LIN {X 0,Y 348.002,Z 736.138,A -85,B 0,C 180,E1 -13689.297,E2 -13689.297} C_VEL
LIN {X 0,Y 349.039,Z 729.917,A -85,B 0,C 180,E1 -13691.322,E2 -13691.322} C_VEL
LIN {X 0,Y 350.021,Z 723.137,A -85,B 0,C 180,E1 -13693.055,E2 -13693.055} C_VEL
LIN {X 0,Y 351.346,Z 714.648,A -85,B 0,C 180,E1 -13694.776,E2 -13694.776} C_VEL
LIN {X 0,Y 352.644,Z 705.984,A -85,B 0,C 180,E1 -13696.201,E2 -13696.201} C_VEL
LIN {X 0,Y 354,Z 696.385,A -85,B 0,C 180,E1 -13697.489,E2 -13697.489} C_VEL
LIN {X 0,Y 355.527,Z 683.397,A -85,B 0,C 180,E1 -13698.887,E2 -13698.887} C_VEL
LIN {X 0,Y 356.754,Z 671.65,A -85,B 0,C 180,E1 -13699.866,E2 -13699.866} C_VEL
LIN {X 0,Y 357.956,Z 658.586,A -85,B 0,C 180,E1 -13700.696,E2 -13700.696} C_VEL
LIN {X 0,Y 358.841,Z 645.608,A -85,B 0,C 180,E1 -13701.281,E2 -13701.281} C_VEL
LIN {X 0,Y 363.919,Z 560.799,A -85,B 0,C 180,E1 -13703.957,E2 -13703.957} C_VEL
LIN {X 0,Y 363.845,Z 556.971,A -85,B 0,C 180,E1 -13704.121,E2 -13704.121} C_VEL
LIN {X 0,Y 360.997,Z 542.499,A -85,B 0,C 180,E1 -13705.115,E2 -13705.115} C_VEL
LIN {X 0,Y 359.502,Z 536.273,A -85,B 0,C 180,E1 -13705.621,E2 -13705.621} C_VEL
LIN {X 0,Y 361.494,Z 519.718,A -85,B 0,C 180,E1 -13708.755,E2 -13708.755} C_VEL
LIN {X 0,Y 360.696,Z 513.547,A -85,B 0,C 180,E1 -13710.252,E2 -13710.252} C_VEL
LIN {X 0,Y 358.682,Z 505.189,A -85,B 0,C 180,E1 -13712.589,E2 -13712.589} C_VEL
LIN {X 0,Y 356.57,Z 498.193,A -85,B 0,C 180,E1 -13714.861,E2 -13714.861} C_VEL
LIN {X 0,Y 353.95,Z 491.68,A -85,B 0,C 180,E1 -13717.415,E2 -13717.415} C_VEL
LIN {X 0,Y 351.895,Z 487.111,A -85,B 0,C 180,E1 -13719.725,E2 -13719.725} C_VEL
LIN {X 0,Y 350.344,Z 483.44,A -85,B 0,C 180,E1 -13722.077,E2 -13722.077} C_VEL
LIN {X 0,Y 348.527,Z 481.325,A -85,B 0,C 180,E1 -13725.107,E2 -13725.107} C_VEL
LIN {X 0,Y 348.251,Z 480.7,A -85,B 0,C 180,E1 -13726.673,E2 -13726.673} C_VEL
LIN {X 0,Y 348.29,Z 480.742,A -85,B 0,C 180,E1 -13728.297,E2 -13728.297} C_VEL
LIN {X 0,Y 348.675,Z 481.499,A -85,B 0,C 180,E1 -13729.991,E2 -13729.991} C_VEL
LIN {X 0,Y 349.596,Z 482.735,A -85,B 0,C 180,E1 -13731.631,E2 -13731.631} C_VEL
LIN {X 0,Y 351.074,Z 484.356,A -85,B 0,C 180,E1 -13733.201,E2 -13733.201} C_VEL
LIN {X 0,Y 352.123,Z 487.497,A -85,B 0,C 180,E1 -13734.632,E2 -13734.632} C_VEL
LIN {X 0,Y 352.81,Z 490.868,A -85,B 0,C 180,E1 -13735.683,E2 -13735.683} C_VEL
LIN {X 0,Y 355.082,Z 501.742,A -85,B 0,C 180,E1 -13738.329,E2 -13738.329} C_VEL
LIN {X 0,Y 357.463,Z 510.29,A -85,B 0,C 180,E1 -13740.056,E2 -13740.056} C_VEL
LIN {X 0,Y 358.938,Z 516.196,A -85,B 0,C 180,E1 -13741.042,E2 -13741.042} C_VEL
LIN {X 0,Y 359.355,Z 523.121,A -85,B 0,C 180,E1 -13741.84,E2 -13741.84} C_VEL
LIN {X 0,Y 359.68,Z 533.701,A -85,B 0,C 180,E1 -13742.9,E2 -13742.9} C_VEL
LIN {X 0,Y 359.381,Z 549.497,A -85,B 0,C 180,E1 -13744.142,E2 -13744.142} C_VEL
LIN {X 0,Y 360.003,Z 556.284,A -85,B 0,C 180,E1 -13744.341,E2 -13744.341} C_VEL
LIN {X 0,Y 357.565,Z 655.14,A -85,B 0,C 180,E1 -13746.468,E2 -13746.468} C_VEL
LIN {X 0,Y 356.73,Z 669.286,A -85,B 0,C 180,E1 -13746.985,E2 -13746.985} C_VEL
LIN {X 0,Y 355.576,Z 683.012,A -85,B 0,C 180,E1 -13747.712,E2 -13747.712} C_VEL
LIN {X 0,Y 354.434,Z 695.886,A -85,B 0,C 180,E1 -13748.631,E2 -13748.631} C_VEL
LIN {X 0,Y 353.249,Z 707.122,A -85,B 0,C 180,E1 -13749.64,E2 -13749.64} C_VEL
LIN {X 0,Y 351.889,Z 718.658,A -85,B 0,C 180,E1 -13750.909,E2 -13750.909} C_VEL
LIN {X 0,Y 350.595,Z 728.367,A -85,B 0,C 180,E1 -13752.198,E2 -13752.198} C_VEL
LIN {X 0,Y 349.238,Z 739.157,A -85,B 0,C 180,E1 -13753.935,E2 -13753.935} C_VEL
LIN {X 0,Y 348.218,Z 747.853,A -85,B 0,C 180,E1 -13755.644,E2 -13755.644} C_VEL
LIN {X 0,Y 347.489,Z 755.405,A -85,B 0,C 180,E1 -13757.441,E2 -13757.441} C_VEL
LIN {X 0,Y 346.772,Z 762.421,A -85,B 0,C 180,E1 -13759.489,E2 -13759.489} C_VEL
LIN {X 0,Y 346.391,Z 768.747,A -85,B 0,C 180,E1 -13761.834,E2 -13761.834} C_VEL
LIN {X 0,Y 346.287,Z 773.108,A -85,B 0,C 180,E1 -13763.971,E2 -13763.971} C_VEL
LIN {X 0,Y 346.266,Z 775.106,A -85,B 0,C 180,E1 -13765.342,E2 -13765.342} C_VEL
LIN {X 0,Y 346.234,Z 776.287,A -85,B 0,C 180,E1 -13766.507,E2 -13766.507} C_VEL
LIN {X 0,Y 346.383,Z 777.549,A -85,B 0,C 180,E1 -13768.836,E2 -13768.836} C_VEL
LIN {X 0,Y 346.383,Z 777.546,A -85,B 0,C 180,E1 -13771.161,E2 -13771.161} C_VEL
LIN {X 0,Y 346.234,Z 776.058,A -85,B 0,C 180,E1 -13773.49,E2 -13773.49} C_VEL
LIN {X 0,Y 346.268,Z 774.768,A -85,B 0,C 180,E1 -13774.655,E2 -13774.655} C_VEL
LIN {X 0,Y 346.323,Z 772.679,A -85,B 0,C 180,E1 -13776.085,E2 -13776.085} C_VEL
LIN {X 0,Y 346.388,Z 768.585,A -85,B 0,C 180,E1 -13778.163,E2 -13778.163} C_VEL
LIN {X 0,Y 346.647,Z 764.085,A -85,B 0,C 180,E1 -13779.922,E2 -13779.922} C_VEL
LIN {X 0,Y 347.28,Z 757.517,A -85,B 0,C 180,E1 -13781.97,E2 -13781.97} C_VEL
LIN {X 0,Y 347.93,Z 750.584,A -85,B 0,C 180,E1 -13783.728,E2 -13783.728} C_VEL
LIN {X 0,Y 348.883,Z 742.235,A -85,B 0,C 180,E1 -13785.479,E2 -13785.479} C_VEL
LIN {X 0,Y 350.113,Z 732.148,A -85,B 0,C 180,E1 -13787.221,E2 -13787.221} C_VEL
LIN {X 0,Y 351.394,Z 722.009,A -85,B 0,C 180,E1 -13788.661,E2 -13788.661} C_VEL
LIN {X 0,Y 352.753,Z 711.083,A -85,B 0,C 180,E1 -13789.944,E2 -13789.944} C_VEL
LIN {X 0,Y 353.991,Z 699.35,A -85,B 0,C 180,E1 -13791.073,E2 -13791.073} C_VEL
LIN {X 0,Y 355.335,Z 686.208,A -85,B 0,C 180,E1 -13792.071,E2 -13792.071} C_VEL
LIN {X 0,Y 356.479,Z 672.058,A -85,B 0,C 180,E1 -13792.875,E2 -13792.875} C_VEL
LIN {X 0,Y 357.403,Z 658.122,A -85,B 0,C 180,E1 -13793.425,E2 -13793.425} C_VEL
LIN {X 0,Y 358.032,Z 637.673,A -85,B 0,C 180,E1 -13793.919,E2 -13793.919} C_VEL
LIN {X 0,Y 359.927,Z 554.026,A -85,B 0,C 180,E1 -13795.701,E2 -13795.701} C_VEL
LIN {X 0,Y 355.225,Z 521.927,A -85,B 0,C 180,E1 -13796.777,E2 -13796.777} C_VEL
LIN {X 0,Y 356.403,Z 514.04,A -85,B 0,C 180,E1 -13798.244,E2 -13798.244} C_VEL
LIN {X 0,Y 355.634,Z 509.249,A -85,B 0,C 180,E1 -13799.261,E2 -13799.261} C_VEL
LIN {X 0,Y 352.934,Z 497.682,A -85,B 0,C 180,E1 -13801.847,E2 -13801.847} C_VEL
LIN {X 0,Y 349.447,Z 484.664,A -85,B 0,C 180,E1 -13804.936,E2 -13804.936} C_VEL
LIN {X 0,Y 347.764,Z 478.78,A -85,B 0,C 180,E1 -13806.471,E2 -13806.471} C_VEL
LIN {X 0,Y 347.786,Z 478.79,A -85,B 0,C 180,E1 -13810.287,E2 -13810.287} C_VEL
LIN {X 0,Y 347.811,Z 478.784,A -85,B 0,C 180,E1 -13813.392,E2 -13813.392} C_VEL
LIN {X 0,Y 347.81,Z 478.786,A -85,B 0,C 180,E1 -13816.669,E2 -13816.669} C_VEL
LIN {X 0,Y 347.777,Z 478.783,A -85,B 0,C 180,E1 -13820.164,E2 -13820.164} C_VEL
LIN {X 0,Y 347.78,Z 478.764,A -85,B 0,C 180,E1 -13824.124,E2 -13824.124} C_VEL
LIN {X 0,Y 347.754,Z 478.787,A -85,B 0,C 180,E1 -13828.301,E2 -13828.301} C_VEL
LIN {X 0,Y 347.796,Z 478.785,A -85,B 0,C 180,E1 -13830.989,E2 -13830.989} C_VEL
LIN {X 0,Y 347.821,Z 478.782,A -85,B 0,C 180,E1 -13833.607,E2 -13833.607} C_VEL
LIN {X 0,Y 347.777,Z 478.774,A -85,B 0,C 180,E1 -13836.161,E2 -13836.161} C_VEL
LIN {X 0,Y 347.796,Z 478.774,A -85,B 0,C 180,E1 -13839.908,E2 -13839.908} C_VEL
LIN {X 0,Y 347.855,Z 478.781,A -85,B 0,C 180,E1 -13842.359,E2 -13842.359} C_VEL
LIN {X 0,Y 347.886,Z 478.773,A -85,B 0,C 180,E1 -13845.97,E2 -13845.97} C_VEL
LIN {X 0,Y 347.922,Z 478.765,A -85,B 0,C 180,E1 -13849.526,E2 -13849.526} C_VEL
LIN {X 0,Y 348.063,Z 478.752,A -85,B 0,C 180,E1 -13851.875,E2 -13851.875} C_VEL
LIN {X 0,Y 348.058,Z 478.744,A -85,B 0,C 180,E1 -13854.206,E2 -13854.206} C_VEL
LIN {X 0,Y 348.198,Z 478.731,A -85,B 0,C 180,E1 -13857.687,E2 -13857.687} C_VEL
LIN {X 0,Y 348.358,Z 478.713,A -85,B 0,C 180,E1 -13860,E2 -13860} C_VEL
LIN {X 0,Y 348.198,Z 478.734,A -85,B 0,C 180,E1 -13862.314,E2 -13862.314} C_VEL
LIN {X 0,Y 348.095,Z 478.746,A -85,B 0,C 180,E1 -13866.958,E2 -13866.958} C_VEL
LIN {X 0,Y 347.958,Z 478.762,A -85,B 0,C 180,E1 -13869.299,E2 -13869.299} C_VEL
LIN {X 0,Y 347.883,Z 478.767,A -85,B 0,C 180,E1 -13872.84,E2 -13872.84} C_VEL
LIN {X 0,Y 347.831,Z 478.782,A -85,B 0,C 180,E1 -13876.432,E2 -13876.432} C_VEL
LIN {X 0,Y 347.846,Z 478.778,A -85,B 0,C 180,E1 -13878.861,E2 -13878.861} C_VEL
LIN {X 0,Y 347.764,Z 478.785,A -85,B 0,C 180,E1 -13882.58,E2 -13882.58} C_VEL
LIN {X 0,Y 347.802,Z 478.783,A -85,B 0,C 180,E1 -13885.109,E2 -13885.109} C_VEL
LIN {X 0,Y 347.803,Z 478.783,A -85,B 0,C 180,E1 -13887.695,E2 -13887.695} C_VEL
LIN {X 0,Y 347.762,Z 478.785,A -85,B 0,C 180,E1 -13890.347,E2 -13890.347} C_VEL
LIN {X 0,Y 347.754,Z 478.786,A -85,B 0,C 180,E1 -13894.049,E2 -13894.049} C_VEL
LIN {X 0,Y 347.756,Z 478.787,A -85,B 0,C 180,E1 -13897.322,E2 -13897.322} C_VEL
LIN {X 0,Y 347.748,Z 478.791,A -85,B 0,C 180,E1 -13900.295,E2 -13900.295} C_VEL
LIN {X 0,Y 347.762,Z 478.789,A -85,B 0,C 180,E1 -13903.402,E2 -13903.402} C_VEL
LIN {X 0,Y 347.779,Z 478.792,A -85,B 0,C 180,E1 -13906.677,E2 -13906.677} C_VEL
LIN {X 0,Y 347.78,Z 478.788,A -85,B 0,C 180,E1 -13910.167,E2 -13910.167} C_VEL
LIN {X 0,Y 347.785,Z 478.785,A -85,B 0,C 180,E1 -13914.127,E2 -13914.127} C_VEL
LIN {X 0,Y 347.774,Z 478.899,A -85,B 0,C 180,E1 -13916.323,E2 -13916.323} C_VEL
LIN {X 0,Y 350.302,Z 488.761,A -85,B 0,C 180,E1 -13919.151,E2 -13919.151} C_VEL
LIN {X 0,Y 352.862,Z 499.54,A -85,B 0,C 180,E1 -13922.094,E2 -13922.094} C_VEL
LIN {X 0,Y 354.273,Z 507.484,A -85,B 0,C 180,E1 -13924.126,E2 -13924.126} C_VEL
LIN {X 0,Y 353.241,Z 516.92,A -85,B 0,C 180,E1 -13926.236,E2 -13926.236} C_VEL
LIN {X 0,Y 358.606,Z 543.403,A -85,B 0,C 180,E1 -13927.182,E2 -13927.182} C_VEL
LIN {X 0,Y 359.417,Z 548.206,A -85,B 0,C 180,E1 -13927.337,E2 -13927.337} C_VEL
LIN {X 0,Y 358.007,Z 631.224,A -85,B 0,C 180,E1 -13928.895,E2 -13928.895} C_VEL
LIN {X 0,Y 357.474,Z 644.098,A -85,B 0,C 180,E1 -13929.352,E2 -13929.352} C_VEL
LIN {X 0,Y 356.593,Z 657.19,A -85,B 0,C 180,E1 -13930.051,E2 -13930.051} C_VEL
LIN {X 0,Y 355.469,Z 669.587,A -85,B 0,C 180,E1 -13930.962,E2 -13930.962} C_VEL
LIN {X 0,Y 354.252,Z 681.206,A -85,B 0,C 180,E1 -13932.093,E2 -13932.093} C_VEL
LIN {X 0,Y 353.116,Z 690.811,A -85,B 0,C 180,E1 -13933.261,E2 -13933.261} C_VEL
LIN {X 0,Y 351.728,Z 700.18,A -85,B 0,C 180,E1 -13934.649,E2 -13934.649} C_VEL
LIN {X 0,Y 350.417,Z 709.509,A -85,B 0,C 180,E1 -13936.371,E2 -13936.371} C_VEL
LIN {X 0,Y 349.322,Z 716.98,A -85,B 0,C 180,E1 -13938.101,E2 -13938.101} C_VEL
LIN {X 0,Y 348.184,Z 723.886,A -85,B 0,C 180,E1 -13940.122,E2 -13940.122} C_VEL
LIN {X 0,Y 347.475,Z 728.531,A -85,B 0,C 180,E1 -13941.862,E2 -13941.862} C_VEL
LIN {X 0,Y 347.067,Z 732.133,A -85,B 0,C 180,E1 -13943.607,E2 -13943.607} C_VEL
LIN {X 0,Y 346.68,Z 734.808,A -85,B 0,C 180,E1 -13945.35,E2 -13945.35} C_VEL
LIN {X 0,Y 346.546,Z 736.986,A -85,B 0,C 180,E1 -13947.677,E2 -13947.677} C_VEL
LIN {X 0,Y 346.395,Z 737.758,A -85,B 0,C 180,E1 -13950.002,E2 -13950.002} C_VEL
LIN {X 0,Y 346.545,Z 737.05,A -85,B 0,C 180,E1 -13952.326,E2 -13952.326} C_VEL
LIN {X 0,Y 346.653,Z 734.923,A -85,B 0,C 180,E1 -13954.653,E2 -13954.653} C_VEL
LIN {X 0,Y 347.06,Z 732.305,A -85,B 0,C 180,E1 -13956.396,E2 -13956.396} C_VEL
LIN {X 0,Y 347.477,Z 728.765,A -85,B 0,C 180,E1 -13958.141,E2 -13958.141} C_VEL
LIN {X 0,Y 348.138,Z 724.186,A -85,B 0,C 180,E1 -13959.882,E2 -13959.882} C_VEL
LIN {X 0,Y 349.206,Z 717.352,A -85,B 0,C 180,E1 -13961.906,E2 -13961.906} C_VEL
LIN {X 0,Y 350.404,Z 709.975,A -85,B 0,C 180,E1 -13963.632,E2 -13963.632} C_VEL
LIN {X 0,Y 351.457,Z 702.468,A -85,B 0,C 180,E1 -13965.069,E2 -13965.069} C_VEL
LIN {X 0,Y 352.73,Z 693.648,A -85,B 0,C 180,E1 -13966.457,E2 -13966.457} C_VEL
LIN {X 0,Y 353.963,Z 683.345,A -85,B 0,C 180,E1 -13967.775,E2 -13967.775} C_VEL
LIN {X 0,Y 355.25,Z 672.22,A -85,B 0,C 180,E1 -13968.903,E2 -13968.903} C_VEL
LIN {X 0,Y 356.257,Z 661.72,A -85,B 0,C 180,E1 -13969.746,E2 -13969.746} C_VEL
LIN {X 0,Y 357.22,Z 649.066,A -85,B 0,C 180,E1 -13970.516,E2 -13970.516} C_VEL
LIN {X 0,Y 357.878,Z 636.708,A -85,B 0,C 180,E1 -13971.041,E2 -13971.041} C_VEL
LIN {X 0,Y 358.257,Z 622.461,A -85,B 0,C 180,E1 -13971.394,E2 -13971.394} C_VEL
LIN {X 0,Y 358.873,Z 586.038,A -85,B 0,C 180,E1 -13972.062,E2 -13972.062} C_VEL
LIN {X 0,Y 358.321,Z 580.227,A -85,B 0,C 180,E1 -13972.214,E2 -13972.214} C_VEL
LIN {X 0,Y 353.289,Z 561.575,A -85,B 0,C 180,E1 -13972.947,E2 -13972.947} C_VEL
LIN {X 0,Y 352.843,Z 555.764,A -85,B 0,C 180,E1 -13973.098,E2 -13973.098} C_VEL
LIN {X 0,Y 352.748,Z 547.495,A -85,B 0,C 180,E1 -13973.274,E2 -13973.274} C_VEL
LIN {X 0,Y 347.839,Z 522.801,A -85,B 0,C 180,E1 -13974.169,E2 -13974.169} C_VEL
LIN {X 0,Y 346.602,Z 516.839,A -85,B 0,C 180,E1 -13974.4,E2 -13974.4} C_VEL
LIN {X 0,Y 347.445,Z 509.457,A -85,B 0,C 180,E1 -13976.102,E2 -13976.102} C_VEL
LIN {X 0,Y 345.815,Z 500.603,A -85,B 0,C 180,E1 -13978.42,E2 -13978.42} C_VEL
LIN {X 0,Y 343.291,Z 489.688,A -85,B 0,C 180,E1 -13981.47,E2 -13981.47} C_VEL
LIN {X 0,Y 340.716,Z 479.667,A -85,B 0,C 180,E1 -13984.476,E2 -13984.476} C_VEL
LIN {X 0,Y 340.718,Z 479.665,A -85,B 0,C 180,E1 -13988.387,E2 -13988.387} C_VEL
LIN {X 0,Y 340.706,Z 479.67,A -85,B 0,C 180,E1 -13992.046,E2 -13992.046} C_VEL
LIN {X 0,Y 340.659,Z 479.676,A -85,B 0,C 180,E1 -13996.227,E2 -13996.227} C_VEL
LIN {X 0,Y 340.695,Z 479.674,A -85,B 0,C 180,E1 -13999.753,E2 -13999.753} C_VEL
LIN {X 0,Y 340.712,Z 479.663,A -85,B 0,C 180,E1 -14003.259,E2 -14003.259} C_VEL
LIN {X 0,Y 340.701,Z 479.672,A -85,B 0,C 180,E1 -14006.154,E2 -14006.154} C_VEL
LIN {X 0,Y 340.717,Z 479.682,A -85,B 0,C 180,E1 -14008.352,E2 -14008.352} C_VEL
LIN {X 0,Y 344.486,Z 495.918,A -85,B 0,C 180,E1 -14011.629,E2 -14011.629} C_VEL
LIN {X 0,Y 346.265,Z 505.327,A -85,B 0,C 180,E1 -14013.479,E2 -14013.479} C_VEL
LIN {X 0,Y 345.11,Z 524.906,A -85,B 0,C 180,E1 -14017.003,E2 -14017.003} C_VEL
LIN {X 0,Y 344.655,Z 531.676,A -85,B 0,C 180,E1 -14018.211,E2 -14018.211} C_VEL
LIN {X 0,Y 347.781,Z 555.235,A -85,B 0,C 180,E1 -14019.034,E2 -14019.034} C_VEL
LIN {X 0,Y 345.289,Z 643.42,A -85,B 0,C 180,E1 -14021.494,E2 -14021.494} C_VEL
LIN {X 0,Y 344.768,Z 655.803,A -85,B 0,C 180,E1 -14022.042,E2 -14022.042} C_VEL
LIN {X 0,Y 344.12,Z 669.789,A -85,B 0,C 180,E1 -14022.927,E2 -14022.927} C_VEL
LIN {X 0,Y 343.327,Z 682.066,A -85,B 0,C 180,E1 -14023.958,E2 -14023.958} C_VEL
LIN {X 0,Y 342.562,Z 694.465,A -85,B 0,C 180,E1 -14025.292,E2 -14025.292} C_VEL
LIN {X 0,Y 341.764,Z 704.362,A -85,B 0,C 180,E1 -14026.624,E2 -14026.624} C_VEL
LIN {X 0,Y 341,Z 713.429,A -85,B 0,C 180,E1 -14028.106,E2 -14028.106} C_VEL
LIN {X 0,Y 340.474,Z 720.954,A -85,B 0,C 180,E1 -14029.594,E2 -14029.594} C_VEL
LIN {X 0,Y 339.947,Z 728.322,A -85,B 0,C 180,E1 -14031.38,E2 -14031.38} C_VEL
LIN {X 0,Y 339.566,Z 734.985,A -85,B 0,C 180,E1 -14033.45,E2 -14033.45} C_VEL
LIN {X 0,Y 339.373,Z 739.411,A -85,B 0,C 180,E1 -14035.248,E2 -14035.248} C_VEL
LIN {X 0,Y 339.25,Z 741.676,A -85,B 0,C 180,E1 -14036.437,E2 -14036.437} C_VEL
LIN {X 0,Y 339.179,Z 743.473,A -85,B 0,C 180,E1 -14037.625,E2 -14037.625} C_VEL
LIN {X 0,Y 339.182,Z 744.84,A -85,B 0,C 180,E1 -14038.813,E2 -14038.813} C_VEL
LIN {X 0,Y 339.194,Z 745.719,A -85,B 0,C 180,E1 -14040,E2 -14040} C_VEL
LIN {X 0,Y 339.298,Z 746.17,A -85,B 0,C 180,E1 -14041.187,E2 -14041.187} C_VEL
LIN {X 0,Y 339.445,Z 746.207,A -85,B 0,C 180,E1 -14042.373,E2 -14042.373} C_VEL
LIN {X 0,Y 339.551,Z 745.781,A -85,B 0,C 180,E1 -14043.56,E2 -14043.56} C_VEL
LIN {X 0,Y 339.598,Z 744.931,A -85,B 0,C 180,E1 -14044.748,E2 -14044.748} C_VEL
LIN {X 0,Y 339.805,Z 743.66,A -85,B 0,C 180,E1 -14045.936,E2 -14045.936} C_VEL
LIN {X 0,Y 340.457,Z 740.793,A -85,B 0,C 180,E1 -14047.747,E2 -14047.747} C_VEL
LIN {X 0,Y 341.06,Z 736.982,A -85,B 0,C 180,E1 -14049.488,E2 -14049.488} C_VEL
LIN {X 0,Y 342,Z 731.922,A -85,B 0,C 180,E1 -14051.258,E2 -14051.258} C_VEL
LIN {X 0,Y 343.04,Z 725.521,A -85,B 0,C 180,E1 -14053.024,E2 -14053.024} C_VEL
LIN {X 0,Y 344.404,Z 717.548,A -85,B 0,C 180,E1 -14054.778,E2 -14054.778} C_VEL
LIN {X 0,Y 345.72,Z 709.388,A -85,B 0,C 180,E1 -14056.231,E2 -14056.231} C_VEL
LIN {X 0,Y 347.283,Z 699.489,A -85,B 0,C 180,E1 -14057.671,E2 -14057.671} C_VEL
LIN {X 0,Y 348.747,Z 688.6,A -85,B 0,C 180,E1 -14058.963,E2 -14058.963} C_VEL
LIN {X 0,Y 349.989,Z 678.066,A -85,B 0,C 180,E1 -14059.96,E2 -14059.96} C_VEL
LIN {X 0,Y 351.248,Z 665.724,A -85,B 0,C 180,E1 -14060.879,E2 -14060.879} C_VEL
LIN {X 0,Y 352.423,Z 651.807,A -85,B 0,C 180,E1 -14061.649,E2 -14061.649} C_VEL
LIN {X 0,Y 353.379,Z 636.861,A -85,B 0,C 180,E1 -14062.202,E2 -14062.202} C_VEL
LIN {X 0,Y 357.783,Z 569.211,A -85,B 0,C 180,E1 -14064.401,E2 -14064.401} C_VEL
LIN {X 0,Y 358.449,Z 559.585,A -85,B 0,C 180,E1 -14064.725,E2 -14064.725} C_VEL
LIN {X 0,Y 355.835,Z 545.585,A -85,B 0,C 180,E1 -14065.719,E2 -14065.719} C_VEL
LIN {X 0,Y 353.816,Z 536.839,A -85,B 0,C 180,E1 -14066.461,E2 -14066.461} C_VEL
LIN {X 0,Y 355.596,Z 523.958,A -85,B 0,C 180,E1 -14068.946,E2 -14068.946} C_VEL
LIN {X 0,Y 355.39,Z 519.767,A -85,B 0,C 180,E1 -14069.909,E2 -14069.909} C_VEL
LIN {X 0,Y 353.845,Z 511.889,A -85,B 0,C 180,E1 -14072.093,E2 -14072.093} C_VEL
LIN {X 0,Y 351.449,Z 503.214,A -85,B 0,C 180,E1 -14074.925,E2 -14074.925} C_VEL
LIN {X 0,Y 349.444,Z 497.813,A -85,B 0,C 180,E1 -14077.111,E2 -14077.111} C_VEL
LIN {X 0,Y 347.397,Z 492.635,A -85,B 0,C 180,E1 -14079.756,E2 -14079.756} C_VEL
LIN {X 0,Y 345.983,Z 489.155,A -85,B 0,C 180,E1 -14082.093,E2 -14082.093} C_VEL
LIN {X 0,Y 344.631,Z 487.472,A -85,B 0,C 180,E1 -14084.458,E2 -14084.458} C_VEL
LIN {X 0,Y 344.284,Z 486.78,A -85,B 0,C 180,E1 -14086.046,E2 -14086.046} C_VEL
LIN {X 0,Y 344.278,Z 486.617,A -85,B 0,C 180,E1 -14087.649,E2 -14087.649} C_VEL
LIN {X 0,Y 344.607,Z 487.101,A -85,B 0,C 180,E1 -14089.259,E2 -14089.259} C_VEL
LIN {X 0,Y 345.342,Z 488.165,A -85,B 0,C 180,E1 -14090.884,E2 -14090.884} C_VEL
LIN {X 0,Y 346.751,Z 489.634,A -85,B 0,C 180,E1 -14092.55,E2 -14092.55} C_VEL
LIN {X 0,Y 347.377,Z 490.657,A -85,B 0,C 180,E1 -14093.243,E2 -14093.243} C_VEL
LIN {X 0,Y 348.313,Z 493.949,A -85,B 0,C 180,E1 -14094.619,E2 -14094.619} C_VEL
LIN {X 0,Y 349.261,Z 499.541,A -85,B 0,C 180,E1 -14096.178,E2 -14096.178} C_VEL
LIN {X 0,Y 351.181,Z 508.468,A -85,B 0,C 180,E1 -14098.308,E2 -14098.308} C_VEL
LIN {X 0,Y 352.743,Z 514.382,A -85,B 0,C 180,E1 -14099.516,E2 -14099.516} C_VEL
LIN {X 0,Y 354.093,Z 520.686,A -85,B 0,C 180,E1 -14100.575,E2 -14100.575} C_VEL
LIN {X 0,Y 354.447,Z 533.188,A -85,B 0,C 180,E1 -14101.97,E2 -14101.97} C_VEL
LIN {X 0,Y 353.828,Z 550.688,A -85,B 0,C 180,E1 -14103.461,E2 -14103.461} C_VEL
LIN {X 0,Y 353.82,Z 555.971,A -85,B 0,C 180,E1 -14103.782,E2 -14103.782} C_VEL
LIN {X 0,Y 353.367,Z 564.545,A -85,B 0,C 180,E1 -14104.051,E2 -14104.051} C_VEL
LIN {X 0,Y 351.037,Z 654.079,A -85,B 0,C 180,E1 -14106.003,E2 -14106.003} C_VEL
LIN {X 0,Y 350.184,Z 668.512,A -85,B 0,C 180,E1 -14106.53,E2 -14106.53} C_VEL
LIN {X 0,Y 349.012,Z 682.364,A -85,B 0,C 180,E1 -14107.269,E2 -14107.269} C_VEL
LIN {X 0,Y 347.875,Z 694.235,A -85,B 0,C 180,E1 -14108.114,E2 -14108.114} C_VEL
LIN {X 0,Y 346.68,Z 705.204,A -85,B 0,C 180,E1 -14109.087,E2 -14109.087} C_VEL
LIN {X 0,Y 345.273,Z 716.969,A -85,B 0,C 180,E1 -14110.374,E2 -14110.374} C_VEL
LIN {X 0,Y 343.746,Z 727.893,A -85,B 0,C 180,E1 -14111.831,E2 -14111.831} C_VEL
LIN {X 0,Y 342.363,Z 738.702,A -85,B 0,C 180,E1 -14113.603,E2 -14113.603} C_VEL
LIN {X 0,Y 341.219,Z 748.018,A -85,B 0,C 180,E1 -14115.477,E2 -14115.477} C_VEL
LIN {X 0,Y 340.394,Z 756.074,A -85,B 0,C 180,E1 -14117.478,E2 -14117.478} C_VEL
LIN {X 0,Y 339.608,Z 763.981,A -85,B 0,C 180,E1 -14119.867,E2 -14119.867} C_VEL
LIN {X 0,Y 339.333,Z 768.737,A -85,B 0,C 180,E1 -14121.662,E2 -14121.662} C_VEL
LIN {X 0,Y 339.223,Z 772.349,A -85,B 0,C 180,E1 -14123.456,E2 -14123.456} C_VEL
LIN {X 0,Y 339.16,Z 774.898,A -85,B 0,C 180,E1 -14125.244,E2 -14125.244} C_VEL
LIN {X 0,Y 339.156,Z 776.03,A -85,B 0,C 180,E1 -14126.434,E2 -14126.434} C_VEL
LIN {X 0,Y 339.303,Z 777.141,A -85,B 0,C 180,E1 -14128.812,E2 -14128.812} C_VEL
LIN {X 0,Y 339.322,Z 777.327,A -85,B 0,C 180,E1 -14129.998,E2 -14129.998} C_VEL
LIN {X 0,Y 339.302,Z 777.137,A -85,B 0,C 180,E1 -14131.185,E2 -14131.185} C_VEL
LIN {X 0,Y 339.155,Z 775.647,A -85,B 0,C 180,E1 -14133.563,E2 -14133.563} C_VEL
LIN {X 0,Y 339.208,Z 772.686,A -85,B 0,C 180,E1 -14135.945,E2 -14135.945} C_VEL
LIN {X 0,Y 339.306,Z 768.165,A -85,B 0,C 180,E1 -14138.335,E2 -14138.335} C_VEL
LIN {X 0,Y 339.605,Z 763.66,A -85,B 0,C 180,E1 -14140.13,E2 -14140.13} C_VEL
LIN {X 0,Y 340.273,Z 757.085,A -85,B 0,C 180,E1 -14142.221,E2 -14142.221} C_VEL
LIN {X 0,Y 340.914,Z 749.508,A -85,B 0,C 180,E1 -14144.166,E2 -14144.166} C_VEL
LIN {X 0,Y 341.968,Z 741.782,A -85,B 0,C 180,E1 -14145.8,E2 -14145.8} C_VEL
LIN {X 0,Y 343.256,Z 731.679,A -85,B 0,C 180,E1 -14147.576,E2 -14147.576} C_VEL
LIN {X 0,Y 344.61,Z 721.52,A -85,B 0,C 180,E1 -14149.043,E2 -14149.043} C_VEL
LIN {X 0,Y 346.18,Z 709.542,A -85,B 0,C 180,E1 -14150.46,E2 -14150.46} C_VEL
LIN {X 0,Y 347.495,Z 697.296,A -85,B 0,C 180,E1 -14151.627,E2 -14151.627} C_VEL
LIN {X 0,Y 348.804,Z 684.434,A -85,B 0,C 180,E1 -14152.585,E2 -14152.585} C_VEL
LIN {X 0,Y 349.967,Z 670.516,A -85,B 0,C 180,E1 -14153.365,E2 -14153.365} C_VEL
LIN {X 0,Y 350.933,Z 655.984,A -85,B 0,C 180,E1 -14153.923,E2 -14153.923} C_VEL
LIN {X 0,Y 351.981,Z 621.161,A -85,B 0,C 180,E1 -14154.71,E2 -14154.71} C_VEL
LIN {X 0,Y 353.45,Z 554.898,A -85,B 0,C 180,E1 -14156.151,E2 -14156.151} C_VEL
LIN {X 0,Y 348.96,Z 524.084,A -85,B 0,C 180,E1 -14157.207,E2 -14157.207} C_VEL
LIN {X 0,Y 348.658,Z 521.666,A -85,B 0,C 180,E1 -14157.326,E2 -14157.326} C_VEL
LIN {X 0,Y 349.606,Z 515.392,A -85,B 0,C 180,E1 -14158.516,E2 -14158.516} C_VEL
LIN {X 0,Y 348.079,Z 507.296,A -85,B 0,C 180,E1 -14160.314,E2 -14160.314} C_VEL
LIN {X 0,Y 344.778,Z 494.153,A -85,B 0,C 180,E1 -14163.39,E2 -14163.39} C_VEL
LIN {X 0,Y 341.241,Z 481.528,A -85,B 0,C 180,E1 -14166.561,E2 -14166.561} C_VEL
LIN {X 0,Y 340.733,Z 479.668,A -85,B 0,C 180,E1 -14167.105,E2 -14167.105} C_VEL
LIN {X 0,Y 340.757,Z 479.665,A -85,B 0,C 180,E1 -14170.261,E2 -14170.261} C_VEL
LIN {X 0,Y 340.771,Z 479.66,A -85,B 0,C 180,E1 -14173.794,E2 -14173.794} C_VEL
LIN {X 0,Y 340.753,Z 479.661,A -85,B 0,C 180,E1 -14177.108,E2 -14177.108} C_VEL
LIN {X 0,Y 340.726,Z 479.661,A -85,B 0,C 180,E1 -14180.251,E2 -14180.251} C_VEL
LIN {X 0,Y 340.703,Z 479.647,A -85,B 0,C 180,E1 -14183.558,E2 -14183.558} C_VEL
LIN {X 0,Y 340.685,Z 479.663,A -85,B 0,C 180,E1 -14186.153,E2 -14186.153} C_VEL
LIN {X 0,Y 340.765,Z 479.662,A -85,B 0,C 180,E1 -14190.332,E2 -14190.332} C_VEL
LIN {X 0,Y 340.795,Z 479.657,A -85,B 0,C 180,E1 -14193.019,E2 -14193.019} C_VEL
LIN {X 0,Y 340.745,Z 479.658,A -85,B 0,C 180,E1 -14195.638,E2 -14195.638} C_VEL
LIN {X 0,Y 340.726,Z 479.649,A -85,B 0,C 180,E1 -14199.473,E2 -14199.473} C_VEL
LIN {X 0,Y 340.846,Z 479.652,A -85,B 0,C 180,E1 -14201.984,E2 -14201.984} C_VEL
LIN {X 0,Y 340.858,Z 479.648,A -85,B 0,C 180,E1 -14205.705,E2 -14205.705} C_VEL
LIN {X 0,Y 340.864,Z 479.644,A -85,B 0,C 180,E1 -14209.306,E2 -14209.306} C_VEL
LIN {X 0,Y 341.065,Z 479.616,A -85,B 0,C 180,E1 -14212.898,E2 -14212.898} C_VEL
LIN {X 0,Y 341.16,Z 479.607,A -85,B 0,C 180,E1 -14217.639,E2 -14217.639} C_VEL
LIN {X 0,Y 341.306,Z 479.591,A -85,B 0,C 180,E1 -14220,E2 -14220} C_VEL
LIN {X 0,Y 341.159,Z 479.609,A -85,B 0,C 180,E1 -14222.361,E2 -14222.361} C_VEL
LIN {X 0,Y 341.064,Z 479.621,A -85,B 0,C 180,E1 -14227.102,E2 -14227.102} C_VEL
LIN {X 0,Y 340.864,Z 479.653,A -85,B 0,C 180,E1 -14230.694,E2 -14230.694} C_VEL
LIN {X 0,Y 340.852,Z 479.645,A -85,B 0,C 180,E1 -14234.326,E2 -14234.326} C_VEL
LIN {X 0,Y 340.828,Z 479.648,A -85,B 0,C 180,E1 -14238.468,E2 -14238.468} C_VEL
LIN {X 0,Y 340.744,Z 479.66,A -85,B 0,C 180,E1 -14241.858,E2 -14241.858} C_VEL
LIN {X 0,Y 340.763,Z 479.659,A -85,B 0,C 180,E1 -14245.665,E2 -14245.665} C_VEL
LIN {X 0,Y 340.733,Z 479.668,A -85,B 0,C 180,E1 -14248.321,E2 -14248.321} C_VEL
LIN {X 0,Y 340.71,Z 479.667,A -85,B 0,C 180,E1 -14251.044,E2 -14251.044} C_VEL
LIN {X 0,Y 340.713,Z 479.669,A -85,B 0,C 180,E1 -14255.28,E2 -14255.28} C_VEL
LIN {X 0,Y 340.711,Z 479.67,A -85,B 0,C 180,E1 -14258.389,E2 -14258.389} C_VEL
LIN {X 0,Y 340.726,Z 479.671,A -85,B 0,C 180,E1 -14262.053,E2 -14262.053} C_VEL
LIN {X 0,Y 340.716,Z 479.667,A -85,B 0,C 180,E1 -14265.47,E2 -14265.47} C_VEL
LIN {X 0,Y 340.72,Z 479.669,A -85,B 0,C 180,E1 -14268.698,E2 -14268.698} C_VEL
LIN {X 0,Y 340.734,Z 479.665,A -85,B 0,C 180,E1 -14271.775,E2 -14271.775} C_VEL
LIN {X 0,Y 340.731,Z 479.729,A -85,B 0,C 180,E1 -14275.711,E2 -14275.711} C_VEL
LIN {X 0,Y 343.49,Z 490.566,A -85,B 0,C 180,E1 -14278.896,E2 -14278.896} C_VEL
LIN {X 0,Y 346.023,Z 501.283,A -85,B 0,C 180,E1 -14281.882,E2 -14281.882} C_VEL
LIN {X 0,Y 347.455,Z 509.021,A -85,B 0,C 180,E1 -14283.902,E2 -14283.902} C_VEL
LIN {X 0,Y 346.567,Z 516.838,A -85,B 0,C 180,E1 -14285.705,E2 -14285.705} C_VEL
LIN {X 0,Y 352.248,Z 544.963,A -85,B 0,C 180,E1 -14286.744,E2 -14286.744} C_VEL
LIN {X 0,Y 352.905,Z 549.798,A -85,B 0,C 180,E1 -14286.892,E2 -14286.892} C_VEL
LIN {X 0,Y 351.481,Z 631.123,A -85,B 0,C 180,E1 -14288.446,E2 -14288.446} C_VEL
LIN {X 0,Y 350.931,Z 644.127,A -85,B 0,C 180,E1 -14288.911,E2 -14288.911} C_VEL
LIN {X 0,Y 350.055,Z 656.719,A -85,B 0,C 180,E1 -14289.586,E2 -14289.586} C_VEL
LIN {X 0,Y 349.005,Z 668.432,A -85,B 0,C 180,E1 -14290.443,E2 -14290.443} C_VEL
LIN {X 0,Y 347.789,Z 679.094,A -85,B 0,C 180,E1 -14291.444,E2 -14291.444} C_VEL
LIN {X 0,Y 346.525,Z 689.747,A -85,B 0,C 180,E1 -14292.709,E2 -14292.709} C_VEL
LIN {X 0,Y 345.182,Z 698.899,A -85,B 0,C 180,E1 -14294.048,E2 -14294.048} C_VEL
LIN {X 0,Y 344.008,Z 707.064,A -85,B 0,C 180,E1 -14295.509,E2 -14295.509} C_VEL
LIN {X 0,Y 342.716,Z 715.076,A -85,B 0,C 180,E1 -14297.266,E2 -14297.266} C_VEL
LIN {X 0,Y 341.871,Z 720.583,A -85,B 0,C 180,E1 -14298.74,E2 -14298.74} C_VEL
LIN {X 0,Y 340.909,Z 725.992,A -85,B 0,C 180,E1 -14300.509,E2 -14300.509} C_VEL
LIN {X 0,Y 340.237,Z 730.754,A -85,B 0,C 180,E1 -14302.526,E2 -14302.526} C_VEL
LIN {X 0,Y 339.857,Z 733.561,A -85,B 0,C 180,E1 -14304.067,E2 -14304.067} C_VEL
LIN {X 0,Y 339.553,Z 736.486,A -85,B 0,C 180,E1 -14306.442,E2 -14306.442} C_VEL
LIN {X 0,Y 339.372,Z 737.956,A -85,B 0,C 180,E1 -14308.815,E2 -14308.815} C_VEL
LIN {X 0,Y 339.372,Z 737.994,A -85,B 0,C 180,E1 -14311.188,E2 -14311.188} C_VEL
LIN {X 0,Y 339.538,Z 736.574,A -85,B 0,C 180,E1 -14313.562,E2 -14313.562} C_VEL
LIN {X 0,Y 339.851,Z 733.711,A -85,B 0,C 180,E1 -14315.936,E2 -14315.936} C_VEL
LIN {X 0,Y 340.239,Z 730.955,A -85,B 0,C 180,E1 -14317.477,E2 -14317.477} C_VEL
LIN {X 0,Y 340.897,Z 726.255,A -85,B 0,C 180,E1 -14319.495,E2 -14319.495} C_VEL
LIN {X 0,Y 341.981,Z 719.927,A -85,B 0,C 180,E1 -14321.56,E2 -14321.56} C_VEL
LIN {X 0,Y 343.069,Z 713.039,A -85,B 0,C 180,E1 -14323.326,E2 -14323.326} C_VEL
LIN {X 0,Y 344.329,Z 704.503,A -85,B 0,C 180,E1 -14325.086,E2 -14325.086} C_VEL
LIN {X 0,Y 345.697,Z 695.78,A -85,B 0,C 180,E1 -14326.537,E2 -14326.537} C_VEL
LIN {X 0,Y 347.112,Z 685.081,A -85,B 0,C 180,E1 -14327.986,E2 -14327.986} C_VEL
LIN {X 0,Y 348.399,Z 674.331,A -85,B 0,C 180,E1 -14329.137,E2 -14329.137} C_VEL
LIN {X 0,Y 349.612,Z 662.324,A -85,B 0,C 180,E1 -14330.138,E2 -14330.138} C_VEL
LIN {X 0,Y 350.626,Z 649.771,A -85,B 0,C 180,E1 -14330.92,E2 -14330.92} C_VEL
LIN {X 0,Y 351.312,Z 637.607,A -85,B 0,C 180,E1 -14331.453,E2 -14331.453} C_VEL
LIN {X 0,Y 351.735,Z 624.046,A -85,B 0,C 180,E1 -14331.811,E2 -14331.811} C_VEL
LIN {X 0,Y 352.843,Z 555.764,A -85,B 0,C 180,E1 -14333.098,E2 -14333.098} C_VEL
LIN {X 0,Y 352.194,Z 551.991,A -85,B 0,C 180,E1 -14333.224,E2 -14333.224} C_VEL
LIN {X 0,Y 350.497,Z 548.579,A -85,B 0,C 180,E1 -14333.422,E2 -14333.422} C_VEL
LIN {X 0,Y 345.542,Z 541.048,A -85,B 0,C 180,E1 -14333.963,E2 -14333.963} C_VEL
LIN {X 0,Y 344.241,Z 537.347,A -85,B 0,C 180,E1 -14334.144,E2 -14334.144} C_VEL
LIN {X 0,Y 339.967,Z 516.885,A -85,B 0,C 180,E1 -14334.947,E2 -14334.947} C_VEL
LIN {X 0,Y 340.627,Z 510.995,A -85,B 0,C 180,E1 -14336.335,E2 -14336.335} C_VEL
LIN {X 0,Y 338.917,Z 501.968,A -85,B 0,C 180,E1 -14338.751,E2 -14338.751} C_VEL
LIN {X 0,Y 336.749,Z 492.506,A -85,B 0,C 180,E1 -14341.451,E2 -14341.451} C_VEL
LIN {X 0,Y 334.018,Z 481.966,A -85,B 0,C 180,E1 -14344.619,E2 -14344.619} C_VEL
LIN {X 0,Y 333.686,Z 480.546,A -85,B 0,C 180,E1 -14345.122,E2 -14345.122} C_VEL
LIN {X 0,Y 333.66,Z 480.544,A -85,B 0,C 180,E1 -14348.799,E2 -14348.799} C_VEL
LIN {X 0,Y 333.639,Z 480.552,A -85,B 0,C 180,E1 -14352.501,E2 -14352.501} C_VEL
LIN {X 0,Y 333.604,Z 480.557,A -85,B 0,C 180,E1 -14355.956,E2 -14355.956} C_VEL
LIN {X 0,Y 333.654,Z 480.547,A -85,B 0,C 180,E1 -14359.316,E2 -14359.316} C_VEL
LIN {X 0,Y 333.672,Z 480.54,A -85,B 0,C 180,E1 -14363.168,E2 -14363.168} C_VEL
LIN {X 0,Y 333.645,Z 480.55,A -85,B 0,C 180,E1 -14366.792,E2 -14366.792} C_VEL
LIN {X 0,Y 333.675,Z 480.659,A -85,B 0,C 180,E1 -14368.052,E2 -14368.052} C_VEL
LIN {X 0,Y 337.462,Z 496.902,A -85,B 0,C 180,E1 -14371.38,E2 -14371.38} C_VEL
LIN {X 0,Y 339.349,Z 506.227,A -85,B 0,C 180,E1 -14373.233,E2 -14373.233} C_VEL
LIN {X 0,Y 338.368,Z 522.531,A -85,B 0,C 180,E1 -14376.212,E2 -14376.212} C_VEL
LIN {X 0,Y 337.765,Z 531.749,A -85,B 0,C 180,E1 -14377.884,E2 -14377.884} C_VEL
LIN {X 0,Y 340.881,Z 556.105,A -85,B 0,C 180,E1 -14378.774,E2 -14378.774} C_VEL
LIN {X 0,Y 338.293,Z 644.516,A -85,B 0,C 180,E1 -14381.333,E2 -14381.333} C_VEL
LIN {X 0,Y 337.677,Z 657.879,A -85,B 0,C 180,E1 -14381.965,E2 -14381.965} C_VEL
LIN {X 0,Y 337.042,Z 671.453,A -85,B 0,C 180,E1 -14382.87,E2 -14382.87} C_VEL
LIN {X 0,Y 336.195,Z 684.429,A -85,B 0,C 180,E1 -14384.025,E2 -14384.025} C_VEL
LIN {X 0,Y 335.432,Z 695.587,A -85,B 0,C 180,E1 -14385.284,E2 -14385.284} C_VEL
LIN {X 0,Y 334.635,Z 705.357,A -85,B 0,C 180,E1 -14386.643,E2 -14386.643} C_VEL
LIN {X 0,Y 333.878,Z 714.345,A -85,B 0,C 180,E1 -14388.157,E2 -14388.157} C_VEL
LIN {X 0,Y 333.34,Z 721.793,A -85,B 0,C 180,E1 -14389.676,E2 -14389.676} C_VEL
LIN {X 0,Y 332.837,Z 729.054,A -85,B 0,C 180,E1 -14391.5,E2 -14391.5} C_VEL
LIN {X 0,Y 332.452,Z 735.377,A -85,B 0,C 180,E1 -14393.511,E2 -14393.511} C_VEL
LIN {X 0,Y 332.297,Z 739.354,A -85,B 0,C 180,E1 -14395.147,E2 -14395.147} C_VEL
LIN {X 0,Y 332.178,Z 741.729,A -85,B 0,C 180,E1 -14396.361,E2 -14396.361} C_VEL
LIN {X 0,Y 332.089,Z 743.585,A -85,B 0,C 180,E1 -14397.574,E2 -14397.574} C_VEL
LIN {X 0,Y 332.084,Z 745.009,A -85,B 0,C 180,E1 -14398.787,E2 -14398.787} C_VEL
LIN {X 0,Y 332.1,Z 745.996,A -85,B 0,C 180,E1 -14400,E2 -14400} C_VEL
LIN {X 0,Y 332.208,Z 746.509,A -85,B 0,C 180,E1 -14401.212,E2 -14401.212} C_VEL
LIN {X 0,Y 332.36,Z 746.605,A -85,B 0,C 180,E1 -14402.424,E2 -14402.424} C_VEL
LIN {X 0,Y 332.472,Z 746.282,A -85,B 0,C 180,E1 -14403.636,E2 -14403.636} C_VEL
LIN {X 0,Y 332.537,Z 745.489,A -85,B 0,C 180,E1 -14404.849,E2 -14404.849} C_VEL
LIN {X 0,Y 332.78,Z 744.269,A -85,B 0,C 180,E1 -14406.061,E2 -14406.061} C_VEL
LIN {X 0,Y 333.444,Z 741.642,A -85,B 0,C 180,E1 -14407.847,E2 -14407.847} C_VEL
LIN {X 0,Y 334.125,Z 737.872,A -85,B 0,C 180,E1 -14409.687,E2 -14409.687} C_VEL
LIN {X 0,Y 335.115,Z 732.959,A -85,B 0,C 180,E1 -14411.492,E2 -14411.492} C_VEL
LIN {X 0,Y 336.219,Z 726.712,A -85,B 0,C 180,E1 -14413.293,E2 -14413.293} C_VEL
LIN {X 0,Y 337.676,Z 718.949,A -85,B 0,C 180,E1 -14415.079,E2 -14415.079} C_VEL
LIN {X 0,Y 339.088,Z 711.059,A -85,B 0,C 180,E1 -14416.558,E2 -14416.558} C_VEL
LIN {X 0,Y 340.738,Z 701.451,A -85,B 0,C 180,E1 -14418.022,E2 -14418.022} C_VEL
LIN {X 0,Y 342.462,Z 689.556,A -85,B 0,C 180,E1 -14419.48,E2 -14419.48} C_VEL
LIN {X 0,Y 343.803,Z 679.323,A -85,B 0,C 180,E1 -14420.491,E2 -14420.491} C_VEL
LIN {X 0,Y 345.168,Z 667.364,A -85,B 0,C 180,E1 -14421.421,E2 -14421.421} C_VEL
LIN {X 0,Y 346.38,Z 654.083,A -85,B 0,C 180,E1 -14422.203,E2 -14422.203} C_VEL
LIN {X 0,Y 347.427,Z 638.929,A -85,B 0,C 180,E1 -14422.799,E2 -14422.799} C_VEL
LIN {X 0,Y 352.98,Z 562.012,A -85,B 0,C 180,E1 -14425.385,E2 -14425.385} C_VEL
LIN {X 0,Y 351.608,Z 552.657,A -85,B 0,C 180,E1 -14426.039,E2 -14426.039} C_VEL
LIN {X 0,Y 348.573,Z 538.905,A -85,B 0,C 180,E1 -14427.219,E2 -14427.219} C_VEL
LIN {X 0,Y 348.3,Z 537.257,A -85,B 0,C 180,E1 -14427.396,E2 -14427.396} C_VEL
LIN {X 0,Y 349.889,Z 526.47,A -85,B 0,C 180,E1 -14429.524,E2 -14429.524} C_VEL
LIN {X 0,Y 349.473,Z 521.601,A -85,B 0,C 180,E1 -14430.763,E2 -14430.763} C_VEL
LIN {X 0,Y 347.892,Z 513.95,A -85,B 0,C 180,E1 -14433.055,E2 -14433.055} C_VEL
LIN {X 0,Y 346.374,Z 508.162,A -85,B 0,C 180,E1 -14435.043,E2 -14435.043} C_VEL
LIN {X 0,Y 344.623,Z 502.87,A -85,B 0,C 180,E1 -14437.311,E2 -14437.311} C_VEL
LIN {X 0,Y 343.138,Z 498.801,A -85,B 0,C 180,E1 -14439.415,E2 -14439.415} C_VEL
LIN {X 0,Y 341.641,Z 494.716,A -85,B 0,C 180,E1 -14442.219,E2 -14442.219} C_VEL
LIN {X 0,Y 340.332,Z 492.872,A -85,B 0,C 180,E1 -14445.402,E2 -14445.402} C_VEL
LIN {X 0,Y 340.454,Z 492.651,A -85,B 0,C 180,E1 -14448,E2 -14448} C_VEL
LIN {X 0,Y 341.295,Z 493.792,A -85,B 0,C 180,E1 -14450.329,E2 -14450.329} C_VEL
LIN {X 0,Y 342.596,Z 495.215,A -85,B 0,C 180,E1 -14452.016,E2 -14452.016} C_VEL
LIN {X 0,Y 343.46,Z 496.378,A -85,B 0,C 180,E1 -14452.942,E2 -14452.942} C_VEL
LIN {X 0,Y 344.295,Z 499.082,A -85,B 0,C 180,E1 -14454.143,E2 -14454.143} C_VEL
LIN {X 0,Y 344.92,Z 503.753,A -85,B 0,C 180,E1 -14455.516,E2 -14455.516} C_VEL
LIN {X 0,Y 346.773,Z 513.278,A -85,B 0,C 180,E1 -14457.857,E2 -14457.857} C_VEL
LIN {X 0,Y 348.189,Z 519.114,A -85,B 0,C 180,E1 -14459.074,E2 -14459.074} C_VEL
LIN {X 0,Y 349.261,Z 524.792,A -85,B 0,C 180,E1 -14460.039,E2 -14460.039} C_VEL
LIN {X 0,Y 349.301,Z 536.871,A -85,B 0,C 180,E1 -14461.407,E2 -14461.407} C_VEL
LIN {X 0,Y 348.456,Z 553.502,A -85,B 0,C 180,E1 -14462.825,E2 -14462.825} C_VEL
LIN {X 0,Y 348.473,Z 558.087,A -85,B 0,C 180,E1 -14463.056,E2 -14463.056} C_VEL
LIN {X 0,Y 346.404,Z 585.561,A -85,B 0,C 180,E1 -14464.029,E2 -14464.029} C_VEL
LIN {X 0,Y 344.486,Z 654.211,A -85,B 0,C 180,E1 -14465.557,E2 -14465.557} C_VEL
LIN {X 0,Y 343.617,Z 668.495,A -85,B 0,C 180,E1 -14466.093,E2 -14466.093} C_VEL
LIN {X 0,Y 342.33,Z 682.842,A -85,B 0,C 180,E1 -14466.88,E2 -14466.88} C_VEL
LIN {X 0,Y 341.151,Z 694.726,A -85,B 0,C 180,E1 -14467.755,E2 -14467.755} C_VEL
LIN {X 0,Y 339.896,Z 705.585,A -85,B 0,C 180,E1 -14468.75,E2 -14468.75} C_VEL
LIN {X 0,Y 338.389,Z 717.668,A -85,B 0,C 180,E1 -14470.116,E2 -14470.116} C_VEL
LIN {X 0,Y 336.951,Z 727.422,A -85,B 0,C 180,E1 -14471.452,E2 -14471.452} C_VEL
LIN {X 0,Y 335.485,Z 738.247,A -85,B 0,C 180,E1 -14473.258,E2 -14473.258} C_VEL
LIN {X 0,Y 334.321,Z 747.3,A -85,B 0,C 180,E1 -14475.107,E2 -14475.107} C_VEL
LIN {X 0,Y 333.3,Z 757.163,A -85,B 0,C 180,E1 -14477.517,E2 -14477.517} C_VEL
LIN {X 0,Y 332.579,Z 764.128,A -85,B 0,C 180,E1 -14479.651,E2 -14479.651} C_VEL
LIN {X 0,Y 332.268,Z 768.759,A -85,B 0,C 180,E1 -14481.484,E2 -14481.484} C_VEL
LIN {X 0,Y 332.163,Z 771.236,A -85,B 0,C 180,E1 -14482.705,E2 -14482.705} C_VEL
LIN {X 0,Y 332.079,Z 773.423,A -85,B 0,C 180,E1 -14484.094,E2 -14484.094} C_VEL
LIN {X 0,Y 332.077,Z 775.794,A -85,B 0,C 180,E1 -14486.358,E2 -14486.358} C_VEL
LIN {X 0,Y 332.208,Z 776.731,A -85,B 0,C 180,E1 -14488.786,E2 -14488.786} C_VEL
LIN {X 0,Y 332.244,Z 776.919,A -85,B 0,C 180,E1 -14489.998,E2 -14489.998} C_VEL
LIN {X 0,Y 332.207,Z 776.727,A -85,B 0,C 180,E1 -14491.211,E2 -14491.211} C_VEL
LIN {X 0,Y 332.078,Z 775.236,A -85,B 0,C 180,E1 -14493.639,E2 -14493.639} C_VEL
LIN {X 0,Y 332.143,Z 772.272,A -85,B 0,C 180,E1 -14496.071,E2 -14496.071} C_VEL
LIN {X 0,Y 332.25,Z 767.746,A -85,B 0,C 180,E1 -14498.513,E2 -14498.513} C_VEL
LIN {X 0,Y 332.55,Z 763.235,A -85,B 0,C 180,E1 -14500.347,E2 -14500.347} C_VEL
LIN {X 0,Y 333.274,Z 756.654,A -85,B 0,C 180,E1 -14502.481,E2 -14502.481} C_VEL
LIN {X 0,Y 334.143,Z 748.429,A -85,B 0,C 180,E1 -14504.617,E2 -14504.617} C_VEL
LIN {X 0,Y 335.255,Z 739.801,A -85,B 0,C 180,E1 -14506.438,E2 -14506.438} C_VEL
LIN {X 0,Y 336.64,Z 729.334,A -85,B 0,C 180,E1 -14508.248,E2 -14508.248} C_VEL
LIN {X 0,Y 338.338,Z 717.57,A -85,B 0,C 180,E1 -14509.884,E2 -14509.884} C_VEL
LIN {X 0,Y 339.821,Z 705.469,A -85,B 0,C 180,E1 -14511.252,E2 -14511.252} C_VEL
LIN {X 0,Y 341.323,Z 692.804,A -85,B 0,C 180,E1 -14512.389,E2 -14512.389} C_VEL
LIN {X 0,Y 342.675,Z 679.24,A -85,B 0,C 180,E1 -14513.332,E2 -14513.332} C_VEL
LIN {X 0,Y 343.79,Z 664.917,A -85,B 0,C 180,E1 -14514.051,E2 -14514.051} C_VEL
LIN {X 0,Y 344.607,Z 650.962,A -85,B 0,C 180,E1 -14514.511,E2 -14514.511} C_VEL
LIN {X 0,Y 346.984,Z 559.717,A -85,B 0,C 180,E1 -14516.525,E2 -14516.525} C_VEL
LIN {X 0,Y 346.826,Z 554.425,A -85,B 0,C 180,E1 -14516.662,E2 -14516.662} C_VEL
LIN {X 0,Y 342.056,Z 521.793,A -85,B 0,C 180,E1 -14517.822,E2 -14517.822} C_VEL
LIN {X 0,Y 342.827,Z 516.782,A -85,B 0,C 180,E1 -14518.798,E2 -14518.798} C_VEL
LIN {X 0,Y 340.544,Z 505.963,A -85,B 0,C 180,E1 -14521.291,E2 -14521.291} C_VEL
LIN {X 0,Y 337.107,Z 492.569,A -85,B 0,C 180,E1 -14524.554,E2 -14524.554} C_VEL
LIN {X 0,Y 333.686,Z 480.542,A -85,B 0,C 180,E1 -14527.74,E2 -14527.74} C_VEL
LIN {X 0,Y 333.692,Z 480.544,A -85,B 0,C 180,E1 -14530.758,E2 -14530.758} C_VEL
LIN {X 0,Y 333.722,Z 480.539,A -85,B 0,C 180,E1 -14534.273,E2 -14534.273} C_VEL
LIN {X 0,Y 333.697,Z 480.538,A -85,B 0,C 180,E1 -14537.627,E2 -14537.627} C_VEL
LIN {X 0,Y 333.674,Z 480.542,A -85,B 0,C 180,E1 -14541.194,E2 -14541.194} C_VEL
LIN {X 0,Y 333.676,Z 480.526,A -85,B 0,C 180,E1 -14545.225,E2 -14545.225} C_VEL
LIN {X 0,Y 333.634,Z 480.546,A -85,B 0,C 180,E1 -14548.222,E2 -14548.222} C_VEL
LIN {X 0,Y 333.702,Z 480.54,A -85,B 0,C 180,E1 -14551.027,E2 -14551.027} C_VEL
LIN {X 0,Y 333.726,Z 480.538,A -85,B 0,C 180,E1 -14553.753,E2 -14553.753} C_VEL
LIN {X 0,Y 333.651,Z 480.515,A -85,B 0,C 180,E1 -14557.719,E2 -14557.719} C_VEL
LIN {X 0,Y 333.782,Z 480.531,A -85,B 0,C 180,E1 -14561.589,E2 -14561.589} C_VEL
LIN {X 0,Y 333.797,Z 480.528,A -85,B 0,C 180,E1 -14565.576,E2 -14565.576} C_VEL
LIN {X 0,Y 333.827,Z 480.519,A -85,B 0,C 180,E1 -14569.078,E2 -14569.078} C_VEL
LIN {X 0,Y 334.015,Z 480.495,A -85,B 0,C 180,E1 -14572.747,E2 -14572.747} C_VEL
LIN {X 0,Y 333.805,Z 480.529,A -85,B 0,C 180,E1 -14575.169,E2 -14575.169} C_VEL
LIN {X 0,Y 334.098,Z 480.487,A -85,B 0,C 180,E1 -14577.589,E2 -14577.589} C_VEL
LIN {X 0,Y 334.257,Z 480.469,A -85,B 0,C 180,E1 -14580,E2 -14580} C_VEL
LIN {X 0,Y 334.097,Z 480.488,A -85,B 0,C 180,E1 -14582.411,E2 -14582.411} C_VEL
LIN {X 0,Y 334.014,Z 480.498,A -85,B 0,C 180,E1 -14587.253,E2 -14587.253} C_VEL
LIN {X 0,Y 333.827,Z 480.527,A -85,B 0,C 180,E1 -14590.922,E2 -14590.922} C_VEL
LIN {X 0,Y 333.798,Z 480.528,A -85,B 0,C 180,E1 -14594.635,E2 -14594.635} C_VEL
LIN {X 0,Y 333.787,Z 480.526,A -85,B 0,C 180,E1 -14598.656,E2 -14598.656} C_VEL
LIN {X 0,Y 333.682,Z 480.538,A -85,B 0,C 180,E1 -14602.279,E2 -14602.279} C_VEL
LIN {X 0,Y 333.726,Z 480.533,A -85,B 0,C 180,E1 -14606.247,E2 -14606.247} C_VEL
LIN {X 0,Y 333.703,Z 480.54,A -85,B 0,C 180,E1 -14608.973,E2 -14608.973} C_VEL
LIN {X 0,Y 333.646,Z 480.549,A -85,B 0,C 180,E1 -14612.591,E2 -14612.591} C_VEL
LIN {X 0,Y 333.669,Z 480.548,A -85,B 0,C 180,E1 -14616.14,E2 -14616.14} C_VEL
LIN {X 0,Y 333.665,Z 480.547,A -85,B 0,C 180,E1 -14619.19,E2 -14619.19} C_VEL
LIN {X 0,Y 333.669,Z 480.547,A -85,B 0,C 180,E1 -14622.51,E2 -14622.51} C_VEL
LIN {X 0,Y 333.663,Z 480.545,A -85,B 0,C 180,E1 -14625.969,E2 -14625.969} C_VEL
LIN {X 0,Y 333.696,Z 480.544,A -85,B 0,C 180,E1 -14629.306,E2 -14629.306} C_VEL
LIN {X 0,Y 333.661,Z 480.536,A -85,B 0,C 180,E1 -14633.169,E2 -14633.169} C_VEL
LIN {X 0,Y 333.693,Z 480.71,A -85,B 0,C 180,E1 -14635.11,E2 -14635.11} C_VEL
LIN {X 0,Y 336.343,Z 490.758,A -85,B 0,C 180,E1 -14638.158,E2 -14638.158} C_VEL
LIN {X 0,Y 338.867,Z 501.56,A -85,B 0,C 180,E1 -14641.25,E2 -14641.25} C_VEL
LIN {X 0,Y 340.622,Z 510.551,A -85,B 0,C 180,E1 -14643.668,E2 -14643.668} C_VEL
LIN {X 0,Y 339.945,Z 516.84,A -85,B 0,C 180,E1 -14645.151,E2 -14645.151} C_VEL
LIN {X 0,Y 345.583,Z 544.806,A -85,B 0,C 180,E1 -14646.228,E2 -14646.228} C_VEL
LIN {X 0,Y 346.45,Z 550.536,A -85,B 0,C 180,E1 -14646.415,E2 -14646.415} C_VEL
LIN {X 0,Y 344.937,Z 632.226,A -85,B 0,C 180,E1 -14648.015,E2 -14648.015} C_VEL
LIN {X 0,Y 344.369,Z 644.928,A -85,B 0,C 180,E1 -14648.489,E2 -14648.489} C_VEL
LIN {X 0,Y 343.455,Z 657.38,A -85,B 0,C 180,E1 -14649.175,E2 -14649.175} C_VEL
LIN {X 0,Y 342.357,Z 669.011,A -85,B 0,C 180,E1 -14650.047,E2 -14650.047} C_VEL
LIN {X 0,Y 341.104,Z 679.621,A -85,B 0,C 180,E1 -14651.066,E2 -14651.066} C_VEL
LIN {X 0,Y 339.737,Z 690.525,A -85,B 0,C 180,E1 -14652.397,E2 -14652.397} C_VEL
LIN {X 0,Y 338.101,Z 701.097,A -85,B 0,C 180,E1 -14654.015,E2 -14654.015} C_VEL
LIN {X 0,Y 336.669,Z 710.392,A -85,B 0,C 180,E1 -14655.803,E2 -14655.803} C_VEL
LIN {X 0,Y 335.429,Z 717.838,A -85,B 0,C 180,E1 -14657.6,E2 -14657.6} C_VEL
LIN {X 0,Y 334.214,Z 724.73,A -85,B 0,C 180,E1 -14659.705,E2 -14659.705} C_VEL
LIN {X 0,Y 333.455,Z 729.364,A -85,B 0,C 180,E1 -14661.518,E2 -14661.518} C_VEL
LIN {X 0,Y 333.012,Z 732.958,A -85,B 0,C 180,E1 -14663.336,E2 -14663.336} C_VEL
LIN {X 0,Y 332.556,Z 735.629,A -85,B 0,C 180,E1 -14665.152,E2 -14665.152} C_VEL
LIN {X 0,Y 332.403,Z 737.805,A -85,B 0,C 180,E1 -14667.578,E2 -14667.578} C_VEL
LIN {X 0,Y 332.274,Z 738.572,A -85,B 0,C 180,E1 -14670.002,E2 -14670.002} C_VEL
LIN {X 0,Y 332.401,Z 737.867,A -85,B 0,C 180,E1 -14672.425,E2 -14672.425} C_VEL
LIN {X 0,Y 332.534,Z 735.742,A -85,B 0,C 180,E1 -14674.851,E2 -14674.851} C_VEL
LIN {X 0,Y 332.983,Z 733.128,A -85,B 0,C 180,E1 -14676.668,E2 -14676.668} C_VEL
LIN {X 0,Y 333.457,Z 729.593,A -85,B 0,C 180,E1 -14678.486,E2 -14678.486} C_VEL
LIN {X 0,Y 334.186,Z 725.023,A -85,B 0,C 180,E1 -14680.299,E2 -14680.299} C_VEL
LIN {X 0,Y 335.337,Z 718.201,A -85,B 0,C 180,E1 -14682.406,E2 -14682.406} C_VEL
LIN {X 0,Y 336.638,Z 710.841,A -85,B 0,C 180,E1 -14684.201,E2 -14684.201} C_VEL
LIN {X 0,Y 337.804,Z 703.357,A -85,B 0,C 180,E1 -14685.693,E2 -14685.693} C_VEL
LIN {X 0,Y 339.157,Z 694.766,A -85,B 0,C 180,E1 -14687.105,E2 -14687.105} C_VEL
LIN {X 0,Y 340.524,Z 684.346,A -85,B 0,C 180,E1 -14688.502,E2 -14688.502} C_VEL
LIN {X 0,Y 341.904,Z 673.302,A -85,B 0,C 180,E1 -14689.671,E2 -14689.671} C_VEL
LIN {X 0,Y 343.214,Z 660.936,A -85,B 0,C 180,E1 -14690.686,E2 -14690.686} C_VEL
LIN {X 0,Y 344.128,Z 649.162,A -85,B 0,C 180,E1 -14691.412,E2 -14691.412} C_VEL
LIN {X 0,Y 344.837,Z 636.537,A -85,B 0,C 180,E1 -14691.955,E2 -14691.955} C_VEL
LIN {X 0,Y 345.252,Z 621.75,A -85,B 0,C 180,E1 -14692.321,E2 -14692.321} C_VEL
LIN {X 0,Y 346.4,Z 549.05,A -85,B 0,C 180,E1 -14693.728,E2 -14693.728} C_VEL
LIN {X 0,Y 344.241,Z 537.347,A -85,B 0,C 180,E1 -14694.144,E2 -14694.144} C_VEL
LIN {X 0,Y 342.92,Z 533.763,A -85,B 0,C 180,E1 -14694.328,E2 -14694.328} C_VEL
LIN {X 0,Y 339.178,Z 528.725,A -85,B 0,C 180,E1 -14694.746,E2 -14694.746} C_VEL
LIN {X 0,Y 335.399,Z 523.706,A -85,B 0,C 180,E1 -14695.178,E2 -14695.178} C_VEL
LIN {X 0,Y 334.02,Z 520.144,A -85,B 0,C 180,E1 -14695.377,E2 -14695.377} C_VEL
LIN {X 0,Y 333.348,Z 516.833,A -85,B 0,C 180,E1 -14695.545,E2 -14695.545} C_VEL
LIN {X 0,Y 333.814,Z 512.555,A -85,B 0,C 180,E1 -14696.577,E2 -14696.577} C_VEL
LIN {X 0,Y 332.023,Z 503.215,A -85,B 0,C 180,E1 -14699.135,E2 -14699.135} C_VEL
LIN {X 0,Y 329.303,Z 491.58,A -85,B 0,C 180,E1 -14702.55,E2 -14702.55} C_VEL
LIN {X 0,Y 326.647,Z 481.42,A -85,B 0,C 180,E1 -14705.754,E2 -14705.754} C_VEL
LIN {X 0,Y 326.619,Z 481.424,A -85,B 0,C 180,E1 -14709.228,E2 -14709.228} C_VEL
LIN {X 0,Y 326.583,Z 481.432,A -85,B 0,C 180,E1 -14712.973,E2 -14712.973} C_VEL
LIN {X 0,Y 326.582,Z 481.425,A -85,B 0,C 180,E1 -14717.029,E2 -14717.029} C_VEL
LIN {X 0,Y 326.618,Z 481.423,A -85,B 0,C 180,E1 -14720.773,E2 -14720.773} C_VEL
LIN {X 0,Y 326.619,Z 481.424,A -85,B 0,C 180,E1 -14724.481,E2 -14724.481} C_VEL
LIN {X 0,Y 326.632,Z 481.534,A -85,B 0,C 180,E1 -14727.732,E2 -14727.732} C_VEL
LIN {X 0,Y 330.793,Z 499.476,A -85,B 0,C 180,E1 -14731.443,E2 -14731.443} C_VEL
LIN {X 0,Y 332.422,Z 507.861,A -85,B 0,C 180,E1 -14733.137,E2 -14733.137} C_VEL
LIN {X 0,Y 331.353,Z 524.679,A -85,B 0,C 180,E1 -14736.235,E2 -14736.235} C_VEL
LIN {X 0,Y 330.853,Z 532.113,A -85,B 0,C 180,E1 -14737.593,E2 -14737.593} C_VEL
LIN {X 0,Y 333.964,Z 556.802,A -85,B 0,C 180,E1 -14738.514,E2 -14738.514} C_VEL
LIN {X 0,Y 331.308,Z 644.549,A -85,B 0,C 180,E1 -14741.125,E2 -14741.125} C_VEL
LIN {X 0,Y 330.709,Z 657.333,A -85,B 0,C 180,E1 -14741.732,E2 -14741.732} C_VEL
LIN {X 0,Y 330.059,Z 671.102,A -85,B 0,C 180,E1 -14742.656,E2 -14742.656} C_VEL
LIN {X 0,Y 329.244,Z 683.203,A -85,B 0,C 180,E1 -14743.73,E2 -14743.73} C_VEL
LIN {X 0,Y 328.418,Z 695.516,A -85,B 0,C 180,E1 -14745.12,E2 -14745.12} C_VEL
LIN {X 0,Y 327.496,Z 706.32,A -85,B 0,C 180,E1 -14746.662,E2 -14746.662} C_VEL
LIN {X 0,Y 326.775,Z 715.203,A -85,B 0,C 180,E1 -14748.21,E2 -14748.21} C_VEL
LIN {X 0,Y 326.135,Z 723.836,A -85,B 0,C 180,E1 -14750.073,E2 -14750.073} C_VEL
LIN {X 0,Y 325.624,Z 730.776,A -85,B 0,C 180,E1 -14751.935,E2 -14751.935} C_VEL
LIN {X 0,Y 325.326,Z 736.299,A -85,B 0,C 180,E1 -14753.799,E2 -14753.799} C_VEL
LIN {X 0,Y 325.167,Z 740.55,A -85,B 0,C 180,E1 -14755.661,E2 -14755.661} C_VEL
LIN {X 0,Y 325.003,Z 743.676,A -85,B 0,C 180,E1 -14757.521,E2 -14757.521} C_VEL
LIN {X 0,Y 324.986,Z 745.168,A -85,B 0,C 180,E1 -14758.761,E2 -14758.761} C_VEL
LIN {X 0,Y 325.005,Z 746.238,A -85,B 0,C 180,E1 -14760,E2 -14760} C_VEL
LIN {X 0,Y 325.118,Z 746.845,A -85,B 0,C 180,E1 -14761.238,E2 -14761.238} C_VEL
LIN {X 0,Y 325.274,Z 747.001,A -85,B 0,C 180,E1 -14762.477,E2 -14762.477} C_VEL
LIN {X 0,Y 325.391,Z 746.752,A -85,B 0,C 180,E1 -14763.715,E2 -14763.715} C_VEL
LIN {X 0,Y 325.481,Z 746.073,A -85,B 0,C 180,E1 -14764.955,E2 -14764.955} C_VEL
LIN {X 0,Y 325.76,Z 744.923,A -85,B 0,C 180,E1 -14766.192,E2 -14766.192} C_VEL
LIN {X 0,Y 326.456,Z 742.47,A -85,B 0,C 180,E1 -14767.982,E2 -14767.982} C_VEL
LIN {X 0,Y 327.199,Z 738.758,A -85,B 0,C 180,E1 -14769.894,E2 -14769.894} C_VEL
LIN {X 0,Y 328.236,Z 733.999,A -85,B 0,C 180,E1 -14771.736,E2 -14771.736} C_VEL
LIN {X 0,Y 329.431,Z 727.993,A -85,B 0,C 180,E1 -14773.572,E2 -14773.572} C_VEL
LIN {X 0,Y 330.971,Z 720.432,A -85,B 0,C 180,E1 -14775.392,E2 -14775.392} C_VEL
LIN {X 0,Y 332.464,Z 712.711,A -85,B 0,C 180,E1 -14776.898,E2 -14776.898} C_VEL
LIN {X 0,Y 334.202,Z 703.467,A -85,B 0,C 180,E1 -14778.387,E2 -14778.387} C_VEL
LIN {X 0,Y 335.982,Z 692.347,A -85,B 0,C 180,E1 -14779.839,E2 -14779.839} C_VEL
LIN {X 0,Y 337.667,Z 680.725,A -85,B 0,C 180,E1 -14781.041,E2 -14781.041} C_VEL
LIN {X 0,Y 339.092,Z 669.081,A -85,B 0,C 180,E1 -14781.985,E2 -14781.985} C_VEL
LIN {X 0,Y 340.531,Z 655.173,A -85,B 0,C 180,E1 -14782.846,E2 -14782.846} C_VEL
LIN {X 0,Y 341.644,Z 640.803,A -85,B 0,C 180,E1 -14783.448,E2 -14783.448} C_VEL
LIN {X 0,Y 346.916,Z 572.253,A -85,B 0,C 180,E1 -14785.826,E2 -14785.826} C_VEL
LIN {X 0,Y 347.653,Z 562.433,A -85,B 0,C 180,E1 -14786.187,E2 -14786.187} C_VEL
LIN {X 0,Y 345.328,Z 548.94,A -85,B 0,C 180,E1 -14787.269,E2 -14787.269} C_VEL
LIN {X 0,Y 342.909,Z 537.941,A -85,B 0,C 180,E1 -14788.336,E2 -14788.336} C_VEL
LIN {X 0,Y 344.266,Z 529.175,A -85,B 0,C 180,E1 -14790.124,E2 -14790.124} C_VEL
LIN {X 0,Y 343.822,Z 524.719,A -85,B 0,C 180,E1 -14791.349,E2 -14791.349} C_VEL
LIN {X 0,Y 342.656,Z 518.637,A -85,B 0,C 180,E1 -14793.244,E2 -14793.244} C_VEL
LIN {X 0,Y 341.018,Z 511.949,A -85,B 0,C 180,E1 -14795.676,E2 -14795.676} C_VEL
LIN {X 0,Y 339.225,Z 506.153,A -85,B 0,C 180,E1 -14798.428,E2 -14798.428} C_VEL
LIN {X 0,Y 338.192,Z 503.352,A -85,B 0,C 180,E1 -14800.107,E2 -14800.107} C_VEL
LIN {X 0,Y 337.472,Z 501.096,A -85,B 0,C 180,E1 -14801.791,E2 -14801.791} C_VEL
LIN {X 0,Y 336.785,Z 499.615,A -85,B 0,C 180,E1 -14803.523,E2 -14803.523} C_VEL
LIN {X 0,Y 336.319,Z 498.488,A -85,B 0,C 180,E1 -14806.4,E2 -14806.4} C_VEL
LIN {X 0,Y 336.809,Z 498.842,A -85,B 0,C 180,E1 -14808.694,E2 -14808.694} C_VEL
LIN {X 0,Y 338.379,Z 500.757,A -85,B 0,C 180,E1 -14811.457,E2 -14811.457} C_VEL
LIN {X 0,Y 339.901,Z 503.059,A -85,B 0,C 180,E1 -14813.156,E2 -14813.156} C_VEL
LIN {X 0,Y 340.492,Z 505.787,A -85,B 0,C 180,E1 -14814.201,E2 -14814.201} C_VEL
LIN {X 0,Y 341.425,Z 513.336,A -85,B 0,C 180,E1 -14816.234,E2 -14816.234} C_VEL
LIN {X 0,Y 343.13,Z 521.453,A -85,B 0,C 180,E1 -14818.128,E2 -14818.128} C_VEL
LIN {X 0,Y 344.4,Z 527.758,A -85,B 0,C 180,E1 -14819.324,E2 -14819.324} C_VEL
LIN {X 0,Y 344.251,Z 539.052,A -85,B 0,C 180,E1 -14820.66,E2 -14820.66} C_VEL
LIN {X 0,Y 343.313,Z 551.87,A -85,B 0,C 180,E1 -14821.828,E2 -14821.828} C_VEL
LIN {X 0,Y 343.43,Z 559.098,A -85,B 0,C 180,E1 -14822.246,E2 -14822.246} C_VEL
LIN {X 0,Y 339.304,Z 607.049,A -85,B 0,C 180,E1 -14824.009,E2 -14824.009} C_VEL
LIN {X 0,Y 337.955,Z 654.317,A -85,B 0,C 180,E1 -14825.094,E2 -14825.094} C_VEL
LIN {X 0,Y 337.058,Z 668.48,A -85,B 0,C 180,E1 -14825.639,E2 -14825.639} C_VEL
LIN {X 0,Y 335.778,Z 682.197,A -85,B 0,C 180,E1 -14826.402,E2 -14826.402} C_VEL
LIN {X 0,Y 334.536,Z 694.153,A -85,B 0,C 180,E1 -14827.291,E2 -14827.291} C_VEL
LIN {X 0,Y 333.117,Z 705.967,A -85,B 0,C 180,E1 -14828.398,E2 -14828.398} C_VEL
LIN {X 0,Y 331.509,Z 718.37,A -85,B 0,C 180,E1 -14829.847,E2 -14829.847} C_VEL
LIN {X 0,Y 329.885,Z 728.944,A -85,B 0,C 180,E1 -14831.362,E2 -14831.362} C_VEL
LIN {X 0,Y 328.194,Z 741.172,A -85,B 0,C 180,E1 -14833.515,E2 -14833.515} C_VEL
LIN {X 0,Y 327.098,Z 750.489,A -85,B 0,C 180,E1 -14835.444,E2 -14835.444} C_VEL
LIN {X 0,Y 326.225,Z 758.598,A -85,B 0,C 180,E1 -14837.557,E2 -14837.557} C_VEL
LIN {X 0,Y 325.569,Z 764.319,A -85,B 0,C 180,E1 -14839.425,E2 -14839.425} C_VEL
LIN {X 0,Y 325.225,Z 768.809,A -85,B 0,C 180,E1 -14841.298,E2 -14841.298} C_VEL
LIN {X 0,Y 325.075,Z 771.184,A -85,B 0,C 180,E1 -14842.545,E2 -14842.545} C_VEL
LIN {X 0,Y 324.975,Z 773.57,A -85,B 0,C 180,E1 -14844.16,E2 -14844.16} C_VEL
LIN {X 0,Y 325,Z 775.532,A -85,B 0,C 180,E1 -14846.279,E2 -14846.279} C_VEL
LIN {X 0,Y 325.113,Z 776.323,A -85,B 0,C 180,E1 -14848.76,E2 -14848.76} C_VEL
LIN {X 0,Y 325.168,Z 776.51,A -85,B 0,C 180,E1 -14849.998,E2 -14849.998} C_VEL
LIN {X 0,Y 325.113,Z 776.318,A -85,B 0,C 180,E1 -14851.237,E2 -14851.237} C_VEL
LIN {X 0,Y 325.004,Z 774.826,A -85,B 0,C 180,E1 -14853.718,E2 -14853.718} C_VEL
LIN {X 0,Y 325.051,Z 771.857,A -85,B 0,C 180,E1 -14856.204,E2 -14856.204} C_VEL
LIN {X 0,Y 325.17,Z 767.327,A -85,B 0,C 180,E1 -14858.7,E2 -14858.7} C_VEL
LIN {X 0,Y 325.512,Z 762.811,A -85,B 0,C 180,E1 -14860.573,E2 -14860.573} C_VEL
LIN {X 0,Y 326.278,Z 756.223,A -85,B 0,C 180,E1 -14862.753,E2 -14862.753} C_VEL
LIN {X 0,Y 327.206,Z 747.99,A -85,B 0,C 180,E1 -14864.935,E2 -14864.935} C_VEL
LIN {X 0,Y 328.396,Z 739.352,A -85,B 0,C 180,E1 -14866.791,E2 -14866.791} C_VEL
LIN {X 0,Y 329.829,Z 728.857,A -85,B 0,C 180,E1 -14868.638,E2 -14868.638} C_VEL
LIN {X 0,Y 331.582,Z 717.068,A -85,B 0,C 180,E1 -14870.307,E2 -14870.307} C_VEL
LIN {X 0,Y 333.049,Z 705.851,A -85,B 0,C 180,E1 -14871.602,E2 -14871.602} C_VEL
LIN {X 0,Y 334.522,Z 693.997,A -85,B 0,C 180,E1 -14872.707,E2 -14872.707} C_VEL
LIN {X 0,Y 335.923,Z 680.865,A -85,B 0,C 180,E1 -14873.666,E2 -14873.666} C_VEL
LIN {X 0,Y 337.128,Z 666.681,A -85,B 0,C 180,E1 -14874.434,E2 -14874.434} C_VEL
LIN {X 0,Y 338.03,Z 652.563,A -85,B 0,C 180,E1 -14874.938,E2 -14874.938} C_VEL
LIN {X 0,Y 340.438,Z 565.308,A -85,B 0,C 180,E1 -14876.902,E2 -14876.902} C_VEL
LIN {X 0,Y 340.456,Z 555.825,A -85,B 0,C 180,E1 -14877.131,E2 -14877.131} C_VEL
LIN {X 0,Y 335.72,Z 523.257,A -85,B 0,C 180,E1 -14878.314,E2 -14878.314} C_VEL
LIN {X 0,Y 335.513,Z 521.696,A -85,B 0,C 180,E1 -14878.385,E2 -14878.385} C_VEL
LIN {X 0,Y 336.002,Z 518.15,A -85,B 0,C 180,E1 -14879.096,E2 -14879.096} C_VEL
LIN {X 0,Y 333.901,Z 508.356,A -85,B 0,C 180,E1 -14881.408,E2 -14881.408} C_VEL
LIN {X 0,Y 330.494,Z 494.951,A -85,B 0,C 180,E1 -14884.754,E2 -14884.754} C_VEL
LIN {X 0,Y 326.632,Z 481.417,A -85,B 0,C 180,E1 -14888.423,E2 -14888.423} C_VEL
LIN {X 0,Y 326.622,Z 481.425,A -85,B 0,C 180,E1 -14891.836,E2 -14891.836} C_VEL
LIN {X 0,Y 326.664,Z 481.417,A -85,B 0,C 180,E1 -14895.23,E2 -14895.23} C_VEL
LIN {X 0,Y 326.624,Z 481.423,A -85,B 0,C 180,E1 -14898.856,E2 -14898.856} C_VEL
LIN {X 0,Y 326.639,Z 481.417,A -85,B 0,C 180,E1 -14901.394,E2 -14901.394} C_VEL
LIN {X 0,Y 326.61,Z 481.401,A -85,B 0,C 180,E1 -14904.85,E2 -14904.85} C_VEL
LIN {X 0,Y 326.606,Z 481.422,A -85,B 0,C 180,E1 -14907.455,E2 -14907.455} C_VEL
LIN {X 0,Y 326.652,Z 481.42,A -85,B 0,C 180,E1 -14910.34,E2 -14910.34} C_VEL
LIN {X 0,Y 326.68,Z 481.418,A -85,B 0,C 180,E1 -14914.516,E2 -14914.516} C_VEL
LIN {X 0,Y 326.61,Z 481.392,A -85,B 0,C 180,E1 -14918.543,E2 -14918.543} C_VEL
LIN {X 0,Y 326.733,Z 481.41,A -85,B 0,C 180,E1 -14921.177,E2 -14921.177} C_VEL
LIN {X 0,Y 326.752,Z 481.406,A -85,B 0,C 180,E1 -14925.433,E2 -14925.433} C_VEL
LIN {X 0,Y 326.763,Z 481.398,A -85,B 0,C 180,E1 -14928.839,E2 -14928.839} C_VEL
LIN {X 0,Y 326.968,Z 481.374,A -85,B 0,C 180,E1 -14932.59,E2 -14932.59} C_VEL
LIN {X 0,Y 326.771,Z 481.406,A -85,B 0,C 180,E1 -14935.065,E2 -14935.065} C_VEL
LIN {X 0,Y 327.038,Z 481.366,A -85,B 0,C 180,E1 -14937.537,E2 -14937.537} C_VEL
LIN {X 0,Y 327.207,Z 481.347,A -85,B 0,C 180,E1 -14940,E2 -14940} C_VEL
LIN {X 0,Y 327.037,Z 481.366,A -85,B 0,C 180,E1 -14942.464,E2 -14942.464} C_VEL
LIN {X 0,Y 326.96,Z 481.378,A -85,B 0,C 180,E1 -14946.676,E2 -14946.676} C_VEL
LIN {X 0,Y 326.805,Z 481.397,A -85,B 0,C 180,E1 -14949.907,E2 -14949.907} C_VEL
LIN {X 0,Y 326.75,Z 481.398,A -85,B 0,C 180,E1 -14953.686,E2 -14953.686} C_VEL
LIN {X 0,Y 326.69,Z 481.407,A -85,B 0,C 180,E1 -14957.529,E2 -14957.529} C_VEL
LIN {X 0,Y 326.655,Z 481.421,A -85,B 0,C 180,E1 -14960.136,E2 -14960.136} C_VEL
LIN {X 0,Y 326.642,Z 481.421,A -85,B 0,C 180,E1 -14964.13,E2 -14964.13} C_VEL
LIN {X 0,Y 326.676,Z 481.412,A -85,B 0,C 180,E1 -14966.859,E2 -14966.859} C_VEL
LIN {X 0,Y 326.633,Z 481.417,A -85,B 0,C 180,E1 -14970.613,E2 -14970.613} C_VEL
LIN {X 0,Y 326.607,Z 481.42,A -85,B 0,C 180,E1 -14974.02,E2 -14974.02} C_VEL
LIN {X 0,Y 326.622,Z 481.419,A -85,B 0,C 180,E1 -14977.241,E2 -14977.241} C_VEL
LIN {X 0,Y 326.597,Z 481.425,A -85,B 0,C 180,E1 -14980.209,E2 -14980.209} C_VEL
LIN {X 0,Y 326.604,Z 481.425,A -85,B 0,C 180,E1 -14983.519,E2 -14983.519} C_VEL
LIN {X 0,Y 326.622,Z 481.426,A -85,B 0,C 180,E1 -14987.02,E2 -14987.02} C_VEL
LIN {X 0,Y 326.64,Z 481.422,A -85,B 0,C 180,E1 -14990.767,E2 -14990.767} C_VEL
LIN {X 0,Y 326.651,Z 481.557,A -85,B 0,C 180,E1 -14994.44,E2 -14994.44} C_VEL
LIN {X 0,Y 329.468,Z 492.262,A -85,B 0,C 180,E1 -14997.775,E2 -14997.775} C_VEL
LIN {X 0,Y 331.954,Z 502.794,A -85,B 0,C 180,E1 -15000.862,E2 -15000.862} C_VEL
LIN {X 0,Y 333.784,Z 512.113,A -85,B 0,C 180,E1 -15003.423,E2 -15003.423} C_VEL
LIN {X 0,Y 333.328,Z 516.943,A -85,B 0,C 180,E1 -15004.595,E2 -15004.595} C_VEL
LIN {X 0,Y 339.195,Z 545.836,A -85,B 0,C 180,E1 -15005.737,E2 -15005.737} C_VEL
LIN {X 0,Y 340.017,Z 551.73,A -85,B 0,C 180,E1 -15005.929,E2 -15005.929} C_VEL
LIN {X 0,Y 338.456,Z 632.127,A -85,B 0,C 180,E1 -15007.532,E2 -15007.532} C_VEL
LIN {X 0,Y 337.863,Z 644.952,A -85,B 0,C 180,E1 -15008.013,E2 -15008.013} C_VEL
LIN {X 0,Y 336.86,Z 658.039,A -85,B 0,C 180,E1 -15008.748,E2 -15008.748} C_VEL
LIN {X 0,Y 335.728,Z 669.588,A -85,B 0,C 180,E1 -15009.636,E2 -15009.636} C_VEL
LIN {X 0,Y 334.41,Z 680.147,A -85,B 0,C 180,E1 -15010.672,E2 -15010.672} C_VEL
LIN {X 0,Y 332.958,Z 691.292,A -85,B 0,C 180,E1 -15012.07,E2 -15012.07} C_VEL
LIN {X 0,Y 331.314,Z 701.554,A -85,B 0,C 180,E1 -15013.678,E2 -15013.678} C_VEL
LIN {X 0,Y 329.81,Z 710.832,A -85,B 0,C 180,E1 -15015.502,E2 -15015.502} C_VEL
LIN {X 0,Y 328.5,Z 718.266,A -85,B 0,C 180,E1 -15017.334,E2 -15017.334} C_VEL
LIN {X 0,Y 327.25,Z 725.151,A -85,B 0,C 180,E1 -15019.484,E2 -15019.484} C_VEL
LIN {X 0,Y 326.435,Z 729.781,A -85,B 0,C 180,E1 -15021.334,E2 -15021.334} C_VEL
LIN {X 0,Y 326.01,Z 732.994,A -85,B 0,C 180,E1 -15022.961,E2 -15022.961} C_VEL
LIN {X 0,Y 325.501,Z 736.039,A -85,B 0,C 180,E1 -15025.047,E2 -15025.047} C_VEL
LIN {X 0,Y 325.318,Z 738.215,A -85,B 0,C 180,E1 -15027.525,E2 -15027.525} C_VEL
LIN {X 0,Y 325.197,Z 738.981,A -85,B 0,C 180,E1 -15030.002,E2 -15030.002} C_VEL
LIN {X 0,Y 325.315,Z 738.276,A -85,B 0,C 180,E1 -15032.478,E2 -15032.478} C_VEL
LIN {X 0,Y 325.48,Z 736.151,A -85,B 0,C 180,E1 -15034.956,E2 -15034.956} C_VEL
LIN {X 0,Y 325.991,Z 733.211,A -85,B 0,C 180,E1 -15037.013,E2 -15037.013} C_VEL
LIN {X 0,Y 326.661,Z 728.633,A -85,B 0,C 180,E1 -15039.287,E2 -15039.287} C_VEL
LIN {X 0,Y 327.555,Z 723.691,A -85,B 0,C 180,E1 -15041.135,E2 -15041.135} C_VEL
LIN {X 0,Y 328.651,Z 717.526,A -85,B 0,C 180,E1 -15042.977,E2 -15042.977} C_VEL
LIN {X 0,Y 329.928,Z 709.877,A -85,B 0,C 180,E1 -15044.812,E2 -15044.812} C_VEL
LIN {X 0,Y 331.584,Z 700.383,A -85,B 0,C 180,E1 -15046.628,E2 -15046.628} C_VEL
LIN {X 0,Y 333.19,Z 689.801,A -85,B 0,C 180,E1 -15048.247,E2 -15048.247} C_VEL
LIN {X 0,Y 334.523,Z 679.655,A -85,B 0,C 180,E1 -15049.484,E2 -15049.484} C_VEL
LIN {X 0,Y 335.868,Z 668.975,A -85,B 0,C 180,E1 -15050.519,E2 -15050.519} C_VEL
LIN {X 0,Y 337.024,Z 657.255,A -85,B 0,C 180,E1 -15051.405,E2 -15051.405} C_VEL
LIN {X 0,Y 337.923,Z 643.89,A -85,B 0,C 180,E1 -15052.147,E2 -15052.147} C_VEL
LIN {X 0,Y 338.557,Z 631.647,A -85,B 0,C 180,E1 -15052.585,E2 -15052.585} C_VEL
LIN {X 0,Y 340.005,Z 550.166,A -85,B 0,C 180,E1 -15054.214,E2 -15054.214} C_VEL
LIN {X 0,Y 335.119,Z 525.248,A -85,B 0,C 180,E1 -15055.168,E2 -15055.168} C_VEL
LIN {X 0,Y 334.02,Z 520.144,A -85,B 0,C 180,E1 -15055.377,E2 -15055.377} C_VEL
LIN {X 0,Y 333.334,Z 517.982,A -85,B 0,C 180,E1 -15055.555,E2 -15055.555} C_VEL
LIN {X 0,Y 331.674,Z 515.265,A -85,B 0,C 180,E1 -15056.094,E2 -15056.094} C_VEL
LIN {X 0,Y 327.658,Z 510.237,A -85,B 0,C 180,E1 -15057.81,E2 -15057.81} C_VEL
LIN {X 0,Y 325.551,Z 505.858,A -85,B 0,C 180,E1 -15059.139,E2 -15059.139} C_VEL
LIN {X 0,Y 324.913,Z 503.525,A -85,B 0,C 180,E1 -15059.808,E2 -15059.808} C_VEL
LIN {X 0,Y 321.973,Z 491.178,A -85,B 0,C 180,E1 -15063.559,E2 -15063.559} C_VEL
LIN {X 0,Y 319.613,Z 482.295,A -85,B 0,C 180,E1 -15066.471,E2 -15066.471} C_VEL
LIN {X 0,Y 319.565,Z 482.306,A -85,B 0,C 180,E1 -15069.669,E2 -15069.669} C_VEL
LIN {X 0,Y 319.528,Z 482.305,A -85,B 0,C 180,E1 -15073.461,E2 -15073.461} C_VEL
LIN {X 0,Y 319.56,Z 482.299,A -85,B 0,C 180,E1 -15077.017,E2 -15077.017} C_VEL
LIN {X 0,Y 319.553,Z 482.303,A -85,B 0,C 180,E1 -15080.371,E2 -15080.371} C_VEL
LIN {X 0,Y 319.586,Z 482.3,A -85,B 0,C 180,E1 -15084.458,E2 -15084.458} C_VEL
LIN {X 0,Y 319.594,Z 482.36,A -85,B 0,C 180,E1 -15087.4,E2 -15087.4} C_VEL
LIN {X 0,Y 323.482,Z 499.106,A -85,B 0,C 180,E1 -15090.912,E2 -15090.912} C_VEL
LIN {X 0,Y 325.506,Z 509.516,A -85,B 0,C 180,E1 -15093.037,E2 -15093.037} C_VEL
LIN {X 0,Y 324.289,Z 527.39,A -85,B 0,C 180,E1 -15096.363,E2 -15096.363} C_VEL
LIN {X 0,Y 323.948,Z 532.573,A -85,B 0,C 180,E1 -15097.304,E2 -15097.304} C_VEL
LIN {X 0,Y 327.063,Z 556.97,A -85,B 0,C 180,E1 -15098.226,E2 -15098.226} C_VEL
LIN {X 0,Y 324.326,Z 644.217,A -85,B 0,C 180,E1 -15100.908,E2 -15100.908} C_VEL
LIN {X 0,Y 323.745,Z 656.466,A -85,B 0,C 180,E1 -15101.489,E2 -15101.489} C_VEL
LIN {X 0,Y 323.052,Z 670.42,A -85,B 0,C 180,E1 -15102.431,E2 -15102.431} C_VEL
LIN {X 0,Y 322.219,Z 682.741,A -85,B 0,C 180,E1 -15103.528,E2 -15103.528} C_VEL
LIN {X 0,Y 321.405,Z 695.192,A -85,B 0,C 180,E1 -15104.95,E2 -15104.95} C_VEL
LIN {X 0,Y 320.557,Z 705.158,A -85,B 0,C 180,E1 -15106.368,E2 -15106.368} C_VEL
LIN {X 0,Y 319.759,Z 714.286,A -85,B 0,C 180,E1 -15107.948,E2 -15107.948} C_VEL
LIN {X 0,Y 319.188,Z 721.861,A -85,B 0,C 180,E1 -15109.534,E2 -15109.534} C_VEL
LIN {X 0,Y 318.666,Z 729.288,A -85,B 0,C 180,E1 -15111.438,E2 -15111.438} C_VEL
LIN {X 0,Y 318.252,Z 736.05,A -85,B 0,C 180,E1 -15113.661,E2 -15113.661} C_VEL
LIN {X 0,Y 318.086,Z 740.475,A -85,B 0,C 180,E1 -15115.565,E2 -15115.565} C_VEL
LIN {X 0,Y 317.92,Z 743.749,A -85,B 0,C 180,E1 -15117.466,E2 -15117.466} C_VEL
LIN {X 0,Y 317.892,Z 745.316,A -85,B 0,C 180,E1 -15118.733,E2 -15118.733} C_VEL
LIN {X 0,Y 317.909,Z 746.448,A -85,B 0,C 180,E1 -15120,E2 -15120} C_VEL
LIN {X 0,Y 318.028,Z 747.164,A -85,B 0,C 180,E1 -15121.266,E2 -15121.266} C_VEL
LIN {X 0,Y 318.189,Z 747.406,A -85,B 0,C 180,E1 -15122.532,E2 -15122.532} C_VEL
LIN {X 0,Y 318.312,Z 747.224,A -85,B 0,C 180,E1 -15123.798,E2 -15123.798} C_VEL
LIN {X 0,Y 318.43,Z 746.634,A -85,B 0,C 180,E1 -15125.065,E2 -15125.065} C_VEL
LIN {X 0,Y 318.742,Z 745.577,A -85,B 0,C 180,E1 -15126.329,E2 -15126.329} C_VEL
LIN {X 0,Y 319.435,Z 743.38,A -85,B 0,C 180,E1 -15128.078,E2 -15128.078} C_VEL
LIN {X 0,Y 320.279,Z 739.713,A -85,B 0,C 180,E1 -15130.11,E2 -15130.11} C_VEL
LIN {X 0,Y 321.373,Z 735.116,A -85,B 0,C 180,E1 -15131.991,E2 -15131.991} C_VEL
LIN {X 0,Y 322.639,Z 729.25,A -85,B 0,C 180,E1 -15133.863,E2 -15133.863} C_VEL
LIN {X 0,Y 324.287,Z 721.964,A -85,B 0,C 180,E1 -15135.718,E2 -15135.718} C_VEL
LIN {X 0,Y 325.889,Z 714.552,A -85,B 0,C 180,E1 -15137.249,E2 -15137.249} C_VEL
LIN {X 0,Y 327.666,Z 705.57,A -85,B 0,C 180,E1 -15138.767,E2 -15138.767} C_VEL
LIN {X 0,Y 329.666,Z 694.545,A -85,B 0,C 180,E1 -15140.276,E2 -15140.276} C_VEL
LIN {X 0,Y 331.355,Z 683.853,A -85,B 0,C 180,E1 -15141.461,E2 -15141.461} C_VEL
LIN {X 0,Y 332.999,Z 672.15,A -85,B 0,C 180,E1 -15142.49,E2 -15142.49} C_VEL
LIN {X 0,Y 334.489,Z 659.124,A -85,B 0,C 180,E1 -15143.365,E2 -15143.365} C_VEL
LIN {X 0,Y 335.683,Z 645.69,A -85,B 0,C 180,E1 -15144.013,E2 -15144.013} C_VEL
LIN {X 0,Y 342.551,Z 564.494,A -85,B 0,C 180,E1 -15146.935,E2 -15146.935} C_VEL
LIN {X 0,Y 340.375,Z 551.304,A -85,B 0,C 180,E1 -15148.046,E2 -15148.046} C_VEL
LIN {X 0,Y 337.747,Z 538.585,A -85,B 0,C 180,E1 -15149.343,E2 -15149.343} C_VEL
LIN {X 0,Y 338.612,Z 533.826,A -85,B 0,C 180,E1 -15150.332,E2 -15150.332} C_VEL
LIN {X 0,Y 338.58,Z 530.258,A -85,B 0,C 180,E1 -15151.261,E2 -15151.261} C_VEL
LIN {X 0,Y 337.399,Z 522.998,A -85,B 0,C 180,E1 -15153.569,E2 -15153.569} C_VEL
LIN {X 0,Y 336.116,Z 517.025,A -85,B 0,C 180,E1 -15155.836,E2 -15155.836} C_VEL
LIN {X 0,Y 334.883,Z 512.471,A -85,B 0,C 180,E1 -15158.004,E2 -15158.004} C_VEL
LIN {X 0,Y 334.021,Z 509.613,A -85,B 0,C 180,E1 -15159.654,E2 -15159.654} C_VEL
LIN {X 0,Y 332.977,Z 506.17,A -85,B 0,C 180,E1 -15162.486,E2 -15162.486} C_VEL
LIN {X 0,Y 332.441,Z 505.036,A -85,B 0,C 180,E1 -15164.238,E2 -15164.238} C_VEL
LIN {X 0,Y 332.373,Z 504.516,A -85,B 0,C 180,E1 -15165.966,E2 -15165.966} C_VEL
LIN {X 0,Y 332.666,Z 504.5,A -85,B 0,C 180,E1 -15167.682,E2 -15167.682} C_VEL
LIN {X 0,Y 333.263,Z 505.218,A -85,B 0,C 180,E1 -15169.392,E2 -15169.392} C_VEL
LIN {X 0,Y 334.374,Z 506.467,A -85,B 0,C 180,E1 -15171.049,E2 -15171.049} C_VEL
LIN {X 0,Y 335.722,Z 508.444,A -85,B 0,C 180,E1 -15172.702,E2 -15172.702} C_VEL
LIN {X 0,Y 336.34,Z 510.738,A -85,B 0,C 180,E1 -15173.69,E2 -15173.69} C_VEL
LIN {X 0,Y 337.44,Z 519.973,A -85,B 0,C 180,E1 -15176.204,E2 -15176.204} C_VEL
LIN {X 0,Y 339.167,Z 528.684,A -85,B 0,C 180,E1 -15178.166,E2 -15178.166} C_VEL
LIN {X 0,Y 339.654,Z 532.613,A -85,B 0,C 180,E1 -15178.848,E2 -15178.848} C_VEL
LIN {X 0,Y 339.208,Z 542.619,A -85,B 0,C 180,E1 -15180.025,E2 -15180.025} C_VEL
LIN {X 0,Y 338.443,Z 552.841,A -85,B 0,C 180,E1 -15180.956,E2 -15180.956} C_VEL
LIN {X 0,Y 338.542,Z 559.949,A -85,B 0,C 180,E1 -15181.394,E2 -15181.394} C_VEL
LIN {X 0,Y 332.233,Z 629.119,A -85,B 0,C 180,E1 -15184.004,E2 -15184.004} C_VEL
LIN {X 0,Y 331.39,Z 655.523,A -85,B 0,C 180,E1 -15184.65,E2 -15184.65} C_VEL
LIN {X 0,Y 330.395,Z 669.97,A -85,B 0,C 180,E1 -15185.241,E2 -15185.241} C_VEL
LIN {X 0,Y 329.059,Z 683.809,A -85,B 0,C 180,E1 -15186.057,E2 -15186.057} C_VEL
LIN {X 0,Y 327.585,Z 697.109,A -85,B 0,C 180,E1 -15187.115,E2 -15187.115} C_VEL
LIN {X 0,Y 326.246,Z 707.373,A -85,B 0,C 180,E1 -15188.142,E2 -15188.142} C_VEL
LIN {X 0,Y 324.278,Z 721.539,A -85,B 0,C 180,E1 -15189.874,E2 -15189.874} C_VEL
LIN {X 0,Y 322.92,Z 731.393,A -85,B 0,C 180,E1 -15191.274,E2 -15191.274} C_VEL
LIN {X 0,Y 321.448,Z 742.098,A -85,B 0,C 180,E1 -15193.159,E2 -15193.159} C_VEL
LIN {X 0,Y 320.405,Z 749.867,A -85,B 0,C 180,E1 -15194.824,E2 -15194.824} C_VEL
LIN {X 0,Y 319.389,Z 757.921,A -85,B 0,C 180,E1 -15196.963,E2 -15196.963} C_VEL
LIN {X 0,Y 318.571,Z 764.536,A -85,B 0,C 180,E1 -15199.19,E2 -15199.19} C_VEL
LIN {X 0,Y 318.162,Z 768.88,A -85,B 0,C 180,E1 -15201.103,E2 -15201.103} C_VEL
LIN {X 0,Y 317.998,Z 771.14,A -85,B 0,C 180,E1 -15202.378,E2 -15202.378} C_VEL
LIN {X 0,Y 317.873,Z 773.631,A -85,B 0,C 180,E1 -15204.226,E2 -15204.226} C_VEL
LIN {X 0,Y 317.923,Z 775.25,A -85,B 0,C 180,E1 -15206.196,E2 -15206.196} C_VEL
LIN {X 0,Y 318.019,Z 775.913,A -85,B 0,C 180,E1 -15208.732,E2 -15208.732} C_VEL
LIN {X 0,Y 318.078,Z 776.101,A -85,B 0,C 180,E1 -15209.998,E2 -15209.998} C_VEL
LIN {X 0,Y 318.018,Z 775.908,A -85,B 0,C 180,E1 -15211.265,E2 -15211.265} C_VEL
LIN {X 0,Y 317.93,Z 774.415,A -85,B 0,C 180,E1 -15213.801,E2 -15213.801} C_VEL
LIN {X 0,Y 317.965,Z 771.442,A -85,B 0,C 180,E1 -15216.343,E2 -15216.343} C_VEL
LIN {X 0,Y 318.107,Z 766.908,A -85,B 0,C 180,E1 -15218.895,E2 -15218.895} C_VEL
LIN {X 0,Y 318.463,Z 762.386,A -85,B 0,C 180,E1 -15220.81,E2 -15220.81} C_VEL
LIN {X 0,Y 319.261,Z 755.791,A -85,B 0,C 180,E1 -15223.039,E2 -15223.039} C_VEL
LIN {X 0,Y 320.126,Z 748.652,A -85,B 0,C 180,E1 -15224.991,E2 -15224.991} C_VEL
LIN {X 0,Y 321.292,Z 740.428,A -85,B 0,C 180,E1 -15226.846,E2 -15226.846} C_VEL
LIN {X 0,Y 322.769,Z 730.278,A -85,B 0,C 180,E1 -15228.732,E2 -15228.732} C_VEL
LIN {X 0,Y 324.575,Z 718.954,A -85,B 0,C 180,E1 -15230.434,E2 -15230.434} C_VEL
LIN {X 0,Y 326.288,Z 706.237,A -85,B 0,C 180,E1 -15231.967,E2 -15231.967} C_VEL
LIN {X 0,Y 327.944,Z 693.416,A -85,B 0,C 180,E1 -15233.188,E2 -15233.188} C_VEL
LIN {X 0,Y 329.4,Z 680.209,A -85,B 0,C 180,E1 -15234.164,E2 -15234.164} C_VEL
LIN {X 0,Y 330.603,Z 666.662,A -85,B 0,C 180,E1 -15234.907,E2 -15234.907} C_VEL
LIN {X 0,Y 331.521,Z 652.735,A -85,B 0,C 180,E1 -15235.42,E2 -15235.42} C_VEL
LIN {X 0,Y 333.175,Z 595.255,A -85,B 0,C 180,E1 -15236.746,E2 -15236.746} C_VEL
LIN {X 0,Y 334.144,Z 557.502,A -85,B 0,C 180,E1 -15237.607,E2 -15237.607} C_VEL
LIN {X 0,Y 329.526,Z 525.121,A -85,B 0,C 180,E1 -15238.809,E2 -15238.809} C_VEL
LIN {X 0,Y 328.983,Z 521.694,A -85,B 0,C 180,E1 -15238.946,E2 -15238.946} C_VEL
LIN {X 0,Y 329.135,Z 519.492,A -85,B 0,C 180,E1 -15239.412,E2 -15239.412} C_VEL
LIN {X 0,Y 327.01,Z 509.784,A -85,B 0,C 180,E1 -15241.77,E2 -15241.77} C_VEL
LIN {X 0,Y 323.874,Z 497.188,A -85,B 0,C 180,E1 -15244.999,E2 -15244.999} C_VEL
LIN {X 0,Y 320.494,Z 485.535,A -85,B 0,C 180,E1 -15248.22,E2 -15248.22} C_VEL
LIN {X 0,Y 319.603,Z 482.294,A -85,B 0,C 180,E1 -15249.186,E2 -15249.186} C_VEL
LIN {X 0,Y 319.618,Z 482.299,A -85,B 0,C 180,E1 -15252.97,E2 -15252.97} C_VEL
LIN {X 0,Y 319.622,Z 482.296,A -85,B 0,C 180,E1 -15256.517,E2 -15256.517} C_VEL
LIN {X 0,Y 319.577,Z 482.294,A -85,B 0,C 180,E1 -15260.375,E2 -15260.375} C_VEL
LIN {X 0,Y 319.551,Z 482.279,A -85,B 0,C 180,E1 -15263.572,E2 -15263.572} C_VEL
LIN {X 0,Y 319.569,Z 482.298,A -85,B 0,C 180,E1 -15266.685,E2 -15266.685} C_VEL
LIN {X 0,Y 319.584,Z 482.297,A -85,B 0,C 180,E1 -15269.616,E2 -15269.616} C_VEL
LIN {X 0,Y 319.599,Z 482.293,A -85,B 0,C 180,E1 -15272.497,E2 -15272.497} C_VEL
LIN {X 0,Y 319.594,Z 482.294,A -85,B 0,C 180,E1 -15275.303,E2 -15275.303} C_VEL
LIN {X 0,Y 319.592,Z 482.276,A -85,B 0,C 180,E1 -15279.4,E2 -15279.4} C_VEL
LIN {X 0,Y 319.647,Z 482.293,A -85,B 0,C 180,E1 -15282.073,E2 -15282.073} C_VEL
LIN {X 0,Y 319.722,Z 482.282,A -85,B 0,C 180,E1 -15286.007,E2 -15286.007} C_VEL
LIN {X 0,Y 319.749,Z 482.275,A -85,B 0,C 180,E1 -15289.873,E2 -15289.873} C_VEL
LIN {X 0,Y 319.922,Z 482.254,A -85,B 0,C 180,E1 -15292.426,E2 -15292.426} C_VEL
LIN {X 0,Y 319.74,Z 482.28,A -85,B 0,C 180,E1 -15294.956,E2 -15294.956} C_VEL
LIN {X 0,Y 319.982,Z 482.245,A -85,B 0,C 180,E1 -15297.483,E2 -15297.483} C_VEL
LIN {X 0,Y 320.159,Z 482.225,A -85,B 0,C 180,E1 -15300,E2 -15300} C_VEL
LIN {X 0,Y 319.981,Z 482.244,A -85,B 0,C 180,E1 -15302.518,E2 -15302.518} C_VEL
LIN {X 0,Y 319.92,Z 482.257,A -85,B 0,C 180,E1 -15306.667,E2 -15306.667} C_VEL
LIN {X 0,Y 319.749,Z 482.278,A -85,B 0,C 180,E1 -15310.128,E2 -15310.128} C_VEL
LIN {X 0,Y 319.72,Z 482.282,A -85,B 0,C 180,E1 -15314.725,E2 -15314.725} C_VEL
LIN {X 0,Y 319.679,Z 482.287,A -85,B 0,C 180,E1 -15319.039,E2 -15319.039} C_VEL
LIN {X 0,Y 319.56,Z 482.302,A -85,B 0,C 180,E1 -15323.32,E2 -15323.32} C_VEL
LIN {X 0,Y 319.625,Z 482.29,A -85,B 0,C 180,E1 -15326.089,E2 -15326.089} C_VEL
LIN {X 0,Y 319.589,Z 482.298,A -85,B 0,C 180,E1 -15328.934,E2 -15328.934} C_VEL
LIN {X 0,Y 319.532,Z 482.306,A -85,B 0,C 180,E1 -15331.862,E2 -15331.862} C_VEL
LIN {X 0,Y 319.575,Z 482.302,A -85,B 0,C 180,E1 -15335.545,E2 -15335.545} C_VEL
LIN {X 0,Y 319.575,Z 482.299,A -85,B 0,C 180,E1 -15338.008,E2 -15338.008} C_VEL
LIN {X 0,Y 319.565,Z 482.305,A -85,B 0,C 180,E1 -15341.608,E2 -15341.608} C_VEL
LIN {X 0,Y 319.572,Z 482.302,A -85,B 0,C 180,E1 -15345.275,E2 -15345.275} C_VEL
LIN {X 0,Y 319.574,Z 482.302,A -85,B 0,C 180,E1 -15348.722,E2 -15348.722} C_VEL
LIN {X 0,Y 319.594,Z 482.29,A -85,B 0,C 180,E1 -15352.341,E2 -15352.341} C_VEL
LIN {X 0,Y 319.608,Z 482.309,A -85,B 0,C 180,E1 -15353.704,E2 -15353.704} C_VEL
LIN {X 0,Y 322.591,Z 493.55,A -85,B 0,C 180,E1 -15357.313,E2 -15357.313} C_VEL
LIN {X 0,Y 325.125,Z 504.346,A -85,B 0,C 180,E1 -15360.545,E2 -15360.545} C_VEL
LIN {X 0,Y 326.941,Z 513.664,A -85,B 0,C 180,E1 -15363.167,E2 -15363.167} C_VEL
LIN {X 0,Y 326.748,Z 516.955,A -85,B 0,C 180,E1 -15363.992,E2 -15363.992} C_VEL
LIN {X 0,Y 332.178,Z 543.727,A -85,B 0,C 180,E1 -15365.102,E2 -15365.102} C_VEL
LIN {X 0,Y 333.614,Z 551.551,A -85,B 0,C 180,E1 -15365.396,E2 -15365.396} C_VEL
LIN {X 0,Y 331.986,Z 632.024,A -85,B 0,C 180,E1 -15367.028,E2 -15367.028} C_VEL
LIN {X 0,Y 331.38,Z 644.973,A -85,B 0,C 180,E1 -15367.519,E2 -15367.519} C_VEL
LIN {X 0,Y 330.417,Z 657.558,A -85,B 0,C 180,E1 -15368.231,E2 -15368.231} C_VEL
LIN {X 0,Y 329.12,Z 670.163,A -85,B 0,C 180,E1 -15369.208,E2 -15369.208} C_VEL
LIN {X 0,Y 327.588,Z 681.964,A -85,B 0,C 180,E1 -15370.417,E2 -15370.417} C_VEL
LIN {X 0,Y 326.188,Z 692.087,A -85,B 0,C 180,E1 -15371.734,E2 -15371.734} C_VEL
LIN {X 0,Y 324.54,Z 702.009,A -85,B 0,C 180,E1 -15373.327,E2 -15373.327} C_VEL
LIN {X 0,Y 322.932,Z 711.272,A -85,B 0,C 180,E1 -15375.186,E2 -15375.186} C_VEL
LIN {X 0,Y 321.594,Z 718.692,A -85,B 0,C 180,E1 -15377.058,E2 -15377.058} C_VEL
LIN {X 0,Y 320.299,Z 725.571,A -85,B 0,C 180,E1 -15379.253,E2 -15379.253} C_VEL
LIN {X 0,Y 319.44,Z 730.196,A -85,B 0,C 180,E1 -15381.143,E2 -15381.143} C_VEL
LIN {X 0,Y 318.945,Z 733.62,A -85,B 0,C 180,E1 -15382.938,E2 -15382.938} C_VEL
LIN {X 0,Y 318.45,Z 736.45,A -85,B 0,C 180,E1 -15384.937,E2 -15384.937} C_VEL
LIN {X 0,Y 318.233,Z 738.625,A -85,B 0,C 180,E1 -15387.47,E2 -15387.47} C_VEL
LIN {X 0,Y 318.123,Z 739.389,A -85,B 0,C 180,E1 -15390.002,E2 -15390.002} C_VEL
LIN {X 0,Y 318.229,Z 738.685,A -85,B 0,C 180,E1 -15392.533,E2 -15392.533} C_VEL
LIN {X 0,Y 318.431,Z 736.56,A -85,B 0,C 180,E1 -15395.066,E2 -15395.066} C_VEL
LIN {X 0,Y 318.926,Z 733.835,A -85,B 0,C 180,E1 -15397.035,E2 -15397.035} C_VEL
LIN {X 0,Y 319.665,Z 729.048,A -85,B 0,C 180,E1 -15399.492,E2 -15399.492} C_VEL
LIN {X 0,Y 320.611,Z 724.109,A -85,B 0,C 180,E1 -15401.38,E2 -15401.38} C_VEL
LIN {X 0,Y 321.737,Z 717.952,A -85,B 0,C 180,E1 -15403.261,E2 -15403.261} C_VEL
LIN {X 0,Y 323.074,Z 710.315,A -85,B 0,C 180,E1 -15405.133,E2 -15405.133} C_VEL
LIN {X 0,Y 324.807,Z 700.832,A -85,B 0,C 180,E1 -15406.986,E2 -15406.986} C_VEL
LIN {X 0,Y 326.452,Z 690.443,A -85,B 0,C 180,E1 -15408.613,E2 -15408.613} C_VEL
LIN {X 0,Y 327.87,Z 680.17,A -85,B 0,C 180,E1 -15409.896,E2 -15409.896} C_VEL
LIN {X 0,Y 329.426,Z 667.783,A -85,B 0,C 180,E1 -15411.102,E2 -15411.102} C_VEL
LIN {X 0,Y 330.653,Z 655.629,A -85,B 0,C 180,E1 -15412.002,E2 -15412.002} C_VEL
LIN {X 0,Y 331.494,Z 643.079,A -85,B 0,C 180,E1 -15412.682,E2 -15412.682} C_VEL
LIN {X 0,Y 332.127,Z 629.888,A -85,B 0,C 180,E1 -15413.13,E2 -15413.13} C_VEL
LIN {X 0,Y 333.653,Z 551.263,A -85,B 0,C 180,E1 -15414.718,E2 -15414.718} C_VEL
LIN {X 0,Y 328.007,Z 522.737,A -85,B 0,C 180,E1 -15415.854,E2 -15415.854} C_VEL
LIN {X 0,Y 326.729,Z 516.999,A -85,B 0,C 180,E1 -15416.111,E2 -15416.111} C_VEL
LIN {X 0,Y 326.84,Z 513.027,A -85,B 0,C 180,E1 -15417.121,E2 -15417.121} C_VEL
LIN {X 0,Y 324.913,Z 503.525,A -85,B 0,C 180,E1 -15419.808,E2 -15419.808} C_VEL
LIN {X 0,Y 323.638,Z 500.748,A -85,B 0,C 180,E1 -15420.698,E2 -15420.698} C_VEL
LIN {X 0,Y 319.816,Z 496.995,A -85,B 0,C 180,E1 -15422.184,E2 -15422.184} C_VEL
LIN {X 0,Y 316.592,Z 494.114,A -85,B 0,C 180,E1 -15423.4,E2 -15423.4} C_VEL
LIN {X 0,Y 314.883,Z 491.632,A -85,B 0,C 180,E1 -15424.337,E2 -15424.337} C_VEL
LIN {X 0,Y 314.555,Z 490.703,A -85,B 0,C 180,E1 -15424.652,E2 -15424.652} C_VEL
LIN {X 0,Y 312.558,Z 483.178,A -85,B 0,C 180,E1 -15427.201,E2 -15427.201} C_VEL
LIN {X 0,Y 312.496,Z 483.181,A -85,B 0,C 180,E1 -15430.71,E2 -15430.71} C_VEL
LIN {X 0,Y 312.458,Z 483.181,A -85,B 0,C 180,E1 -15434.21,E2 -15434.21} C_VEL
LIN {X 0,Y 312.49,Z 483.175,A -85,B 0,C 180,E1 -15437.919,E2 -15437.919} C_VEL
LIN {X 0,Y 312.505,Z 483.177,A -85,B 0,C 180,E1 -15440.972,E2 -15440.972} C_VEL
LIN {X 0,Y 312.539,Z 483.179,A -85,B 0,C 180,E1 -15444.221,E2 -15444.221} C_VEL
LIN {X 0,Y 312.583,Z 483.36,A -85,B 0,C 180,E1 -15447.085,E2 -15447.085} C_VEL
LIN {X 0,Y 316.59,Z 500.643,A -85,B 0,C 180,E1 -15450.766,E2 -15450.766} C_VEL
LIN {X 0,Y 318.512,Z 510.242,A -85,B 0,C 180,E1 -15452.751,E2 -15452.751} C_VEL
LIN {X 0,Y 317.734,Z 522.89,A -85,B 0,C 180,E1 -15455.148,E2 -15455.148} C_VEL
LIN {X 0,Y 317.058,Z 532.729,A -85,B 0,C 180,E1 -15456.99,E2 -15456.99} C_VEL
LIN {X 0,Y 320.126,Z 558.141,A -85,B 0,C 180,E1 -15457.971,E2 -15457.971} C_VEL
LIN {X 0,Y 317.292,Z 645.489,A -85,B 0,C 180,E1 -15460.763,E2 -15460.763} C_VEL
LIN {X 0,Y 316.622,Z 659.316,A -85,B 0,C 180,E1 -15461.476,E2 -15461.476} C_VEL
LIN {X 0,Y 315.98,Z 671.694,A -85,B 0,C 180,E1 -15462.359,E2 -15462.359} C_VEL
LIN {X 0,Y 315.089,Z 684.54,A -85,B 0,C 180,E1 -15463.562,E2 -15463.562} C_VEL
LIN {X 0,Y 314.243,Z 696.085,A -85,B 0,C 180,E1 -15464.93,E2 -15464.93} C_VEL
LIN {X 0,Y 313.411,Z 705.956,A -85,B 0,C 180,E1 -15466.381,E2 -15466.381} C_VEL
LIN {X 0,Y 312.63,Z 715.033,A -85,B 0,C 180,E1 -15467.998,E2 -15467.998} C_VEL
LIN {X 0,Y 312.062,Z 722.562,A -85,B 0,C 180,E1 -15469.62,E2 -15469.62} C_VEL
LIN {X 0,Y 311.533,Z 729.914,A -85,B 0,C 180,E1 -15471.568,E2 -15471.568} C_VEL
LIN {X 0,Y 311.18,Z 735.967,A -85,B 0,C 180,E1 -15473.596,E2 -15473.596} C_VEL
LIN {X 0,Y 311.006,Z 740.322,A -85,B 0,C 180,E1 -15475.463,E2 -15475.463} C_VEL
LIN {X 0,Y 310.841,Z 743.736,A -85,B 0,C 180,E1 -15477.408,E2 -15477.408} C_VEL
LIN {X 0,Y 310.801,Z 745.437,A -85,B 0,C 180,E1 -15478.704,E2 -15478.704} C_VEL
LIN {X 0,Y 310.814,Z 746.648,A -85,B 0,C 180,E1 -15480,E2 -15480} C_VEL
LIN {X 0,Y 310.935,Z 747.437,A -85,B 0,C 180,E1 -15481.295,E2 -15481.295} C_VEL
LIN {X 0,Y 311.103,Z 747.802,A -85,B 0,C 180,E1 -15482.589,E2 -15482.589} C_VEL
LIN {X 0,Y 311.233,Z 747.693,A -85,B 0,C 180,E1 -15483.884,E2 -15483.884} C_VEL
LIN {X 0,Y 311.383,Z 747.176,A -85,B 0,C 180,E1 -15485.18,E2 -15485.18} C_VEL
LIN {X 0,Y 311.728,Z 746.243,A -85,B 0,C 180,E1 -15486.472,E2 -15486.472} C_VEL
LIN {X 0,Y 312.417,Z 744.272,A -85,B 0,C 180,E1 -15488.18,E2 -15488.18} C_VEL
LIN {X 0,Y 313.364,Z 740.678,A -85,B 0,C 180,E1 -15490.336,E2 -15490.336} C_VEL
LIN {X 0,Y 314.52,Z 736.243,A -85,B 0,C 180,E1 -15492.256,E2 -15492.256} C_VEL
LIN {X 0,Y 315.883,Z 730.608,A -85,B 0,C 180,E1 -15494.166,E2 -15494.166} C_VEL
LIN {X 0,Y 317.641,Z 723.528,A -85,B 0,C 180,E1 -15496.055,E2 -15496.055} C_VEL
LIN {X 0,Y 319.304,Z 716.326,A -85,B 0,C 180,E1 -15497.616,E2 -15497.616} C_VEL
LIN {X 0,Y 321.448,Z 706.603,A -85,B 0,C 180,E1 -15499.339,E2 -15499.339} C_VEL
LIN {X 0,Y 323.57,Z 695.8,A -85,B 0,C 180,E1 -15500.875,E2 -15500.875} C_VEL
LIN {X 0,Y 325.562,Z 684.087,A -85,B 0,C 180,E1 -15502.196,E2 -15502.196} C_VEL
LIN {X 0,Y 327.305,Z 672.442,A -85,B 0,C 180,E1 -15503.238,E2 -15503.238} C_VEL
LIN {X 0,Y 328.929,Z 659.611,A -85,B 0,C 180,E1 -15504.119,E2 -15504.119} C_VEL
LIN {X 0,Y 330.277,Z 645.676,A -85,B 0,C 180,E1 -15504.809,E2 -15504.809} C_VEL
LIN {X 0,Y 336.474,Z 576.809,A -85,B 0,C 180,E1 -15507.356,E2 -15507.356} C_VEL
LIN {X 0,Y 337.471,Z 565.977,A -85,B 0,C 180,E1 -15507.772,E2 -15507.772} C_VEL
LIN {X 0,Y 335.809,Z 554.641,A -85,B 0,C 180,E1 -15508.774,E2 -15508.774} C_VEL
LIN {X 0,Y 333.327,Z 541.732,A -85,B 0,C 180,E1 -15510.142,E2 -15510.142} C_VEL
LIN {X 0,Y 332.851,Z 539.164,A -85,B 0,C 180,E1 -15510.447,E2 -15510.447} C_VEL
LIN {X 0,Y 333.312,Z 535.869,A -85,B 0,C 180,E1 -15511.191,E2 -15511.191} C_VEL
LIN {X 0,Y 332.542,Z 529.08,A -85,B 0,C 180,E1 -15513.332,E2 -15513.332} C_VEL
LIN {X 0,Y 331.593,Z 523.603,A -85,B 0,C 180,E1 -15515.385,E2 -15515.385} C_VEL
LIN {X 0,Y 330.247,Z 517.844,A -85,B 0,C 180,E1 -15518.108,E2 -15518.108} C_VEL
LIN {X 0,Y 329.552,Z 514.99,A -85,B 0,C 180,E1 -15519.847,E2 -15519.847} C_VEL
LIN {X 0,Y 328.915,Z 512.875,A -85,B 0,C 180,E1 -15521.594,E2 -15521.594} C_VEL
LIN {X 0,Y 328.545,Z 511.353,A -85,B 0,C 180,E1 -15523.338,E2 -15523.338} C_VEL
LIN {X 0,Y 328.314,Z 510.589,A -85,B 0,C 180,E1 -15525.055,E2 -15525.055} C_VEL
LIN {X 0,Y 328.541,Z 510.39,A -85,B 0,C 180,E1 -15526.8,E2 -15526.8} C_VEL
LIN {X 0,Y 329.059,Z 510.788,A -85,B 0,C 180,E1 -15528.539,E2 -15528.539} C_VEL
LIN {X 0,Y 330.049,Z 511.911,A -85,B 0,C 180,E1 -15530.295,E2 -15530.295} C_VEL
LIN {X 0,Y 331.445,Z 513.71,A -85,B 0,C 180,E1 -15532.052,E2 -15532.052} C_VEL
LIN {X 0,Y 332.03,Z 514.762,A -85,B 0,C 180,E1 -15532.753,E2 -15532.753} C_VEL
LIN {X 0,Y 332.372,Z 517.444,A -85,B 0,C 180,E1 -15533.695,E2 -15533.695} C_VEL
LIN {X 0,Y 333.263,Z 525.595,A -85,B 0,C 180,E1 -15535.895,E2 -15535.895} C_VEL
LIN {X 0,Y 334.746,Z 533.629,A -85,B 0,C 180,E1 -15537.723,E2 -15537.723} C_VEL
LIN {X 0,Y 334.937,Z 536.421,A -85,B 0,C 180,E1 -15538.2,E2 -15538.2} C_VEL
LIN {X 0,Y 334.42,Z 544.589,A -85,B 0,C 180,E1 -15539.197,E2 -15539.197} C_VEL
LIN {X 0,Y 333.683,Z 552.126,A -85,B 0,C 180,E1 -15539.914,E2 -15539.914} C_VEL
LIN {X 0,Y 333.841,Z 561.355,A -85,B 0,C 180,E1 -15540.516,E2 -15540.516} C_VEL
LIN {X 0,Y 325.141,Z 650.695,A -85,B 0,C 180,E1 -15543.998,E2 -15543.998} C_VEL
LIN {X 0,Y 324.243,Z 665.339,A -85,B 0,C 180,E1 -15544.524,E2 -15544.524} C_VEL
LIN {X 0,Y 322.801,Z 681.334,A -85,B 0,C 180,E1 -15545.392,E2 -15545.392} C_VEL
LIN {X 0,Y 321.477,Z 694.354,A -85,B 0,C 180,E1 -15546.314,E2 -15546.314} C_VEL
LIN {X 0,Y 320.018,Z 706.794,A -85,B 0,C 180,E1 -15547.454,E2 -15547.454} C_VEL
LIN {X 0,Y 318.357,Z 719.789,A -85,B 0,C 180,E1 -15548.976,E2 -15548.976} C_VEL
LIN {X 0,Y 316.769,Z 729.795,A -85,B 0,C 180,E1 -15550.391,E2 -15550.391} C_VEL
LIN {X 0,Y 315.223,Z 739.831,A -85,B 0,C 180,E1 -15552.146,E2 -15552.146} C_VEL
LIN {X 0,Y 313.87,Z 748.879,A -85,B 0,C 180,E1 -15554.078,E2 -15554.078} C_VEL
LIN {X 0,Y 312.816,Z 756.228,A -85,B 0,C 180,E1 -15556.022,E2 -15556.022} C_VEL
LIN {X 0,Y 311.773,Z 763.098,A -85,B 0,C 180,E1 -15558.293,E2 -15558.293} C_VEL
LIN {X 0,Y 311.237,Z 767.656,A -85,B 0,C 180,E1 -15560.248,E2 -15560.248} C_VEL
LIN {X 0,Y 310.943,Z 771.122,A -85,B 0,C 180,E1 -15562.204,E2 -15562.204} C_VEL
LIN {X 0,Y 310.789,Z 773.658,A -85,B 0,C 180,E1 -15564.262,E2 -15564.262} C_VEL
LIN {X 0,Y 310.825,Z 774.975,A -85,B 0,C 180,E1 -15566.109,E2 -15566.109} C_VEL
LIN {X 0,Y 310.925,Z 775.503,A -85,B 0,C 180,E1 -15568.703,E2 -15568.703} C_VEL
LIN {X 0,Y 310.989,Z 775.692,A -85,B 0,C 180,E1 -15569.998,E2 -15569.998} C_VEL
LIN {X 0,Y 310.923,Z 775.498,A -85,B 0,C 180,E1 -15571.294,E2 -15571.294} C_VEL
LIN {X 0,Y 310.857,Z 774.005,A -85,B 0,C 180,E1 -15573.887,E2 -15573.887} C_VEL
LIN {X 0,Y 310.89,Z 771.028,A -85,B 0,C 180,E1 -15576.488,E2 -15576.488} C_VEL
LIN {X 0,Y 311.061,Z 766.491,A -85,B 0,C 180,E1 -15579.098,E2 -15579.098} C_VEL
LIN {X 0,Y 311.435,Z 761.963,A -85,B 0,C 180,E1 -15581.057,E2 -15581.057} C_VEL
LIN {X 0,Y 312.245,Z 755.359,A -85,B 0,C 180,E1 -15583.337,E2 -15583.337} C_VEL
LIN {X 0,Y 313.065,Z 748.976,A -85,B 0,C 180,E1 -15585.137,E2 -15585.137} C_VEL
LIN {X 0,Y 314.447,Z 739.98,A -85,B 0,C 180,E1 -15587.224,E2 -15587.224} C_VEL
LIN {X 0,Y 315.998,Z 729.815,A -85,B 0,C 180,E1 -15589.149,E2 -15589.149} C_VEL
LIN {X 0,Y 317.845,Z 718.457,A -85,B 0,C 180,E1 -15590.886,E2 -15590.886} C_VEL
LIN {X 0,Y 319.498,Z 706.941,A -85,B 0,C 180,E1 -15592.313,E2 -15592.313} C_VEL
LIN {X 0,Y 321.173,Z 694.613,A -85,B 0,C 180,E1 -15593.536,E2 -15593.536} C_VEL
LIN {X 0,Y 322.778,Z 680.681,A -85,B 0,C 180,E1 -15594.607,E2 -15594.607} C_VEL
LIN {X 0,Y 324.105,Z 666.638,A -85,B 0,C 180,E1 -15595.398,E2 -15595.398} C_VEL
LIN {X 0,Y 325.057,Z 652.906,A -85,B 0,C 180,E1 -15595.92,E2 -15595.92} C_VEL
LIN {X 0,Y 327.68,Z 565,A -85,B 0,C 180,E1 -15597.968,E2 -15597.968} C_VEL
LIN {X 0,Y 327.61,Z 556.842,A -85,B 0,C 180,E1 -15598.183,E2 -15598.183} C_VEL
LIN {X 0,Y 322.72,Z 523.094,A -85,B 0,C 180,E1 -15599.483,E2 -15599.483} C_VEL
LIN {X 0,Y 322.395,Z 521.48,A -85,B 0,C 180,E1 -15599.59,E2 -15599.59} C_VEL
LIN {X 0,Y 320.156,Z 511.262,A -85,B 0,C 180,E1 -15602.134,E2 -15602.134} C_VEL
LIN {X 0,Y 317.329,Z 499.782,A -85,B 0,C 180,E1 -15605.155,E2 -15605.155} C_VEL
LIN {X 0,Y 314.006,Z 488.21,A -85,B 0,C 180,E1 -15608.431,E2 -15608.431} C_VEL
LIN {X 0,Y 312.546,Z 483.18,A -85,B 0,C 180,E1 -15609.959,E2 -15609.959} C_VEL
LIN {X 0,Y 312.587,Z 483.171,A -85,B 0,C 180,E1 -15614.183,E2 -15614.183} C_VEL
LIN {X 0,Y 312.548,Z 483.171,A -85,B 0,C 180,E1 -15617.903,E2 -15617.903} C_VEL
LIN {X 0,Y 312.55,Z 483.172,A -85,B 0,C 180,E1 -15621.904,E2 -15621.904} C_VEL
LIN {X 0,Y 312.497,Z 483.171,A -85,B 0,C 180,E1 -15625.789,E2 -15625.789} C_VEL
LIN {X 0,Y 312.518,Z 483.174,A -85,B 0,C 180,E1 -15628.853,E2 -15628.853} C_VEL
LIN {X 0,Y 312.565,Z 483.17,A -85,B 0,C 180,E1 -15631.824,E2 -15631.824} C_VEL
LIN {X 0,Y 312.575,Z 483.172,A -85,B 0,C 180,E1 -15634.71,E2 -15634.71} C_VEL
LIN {X 0,Y 312.528,Z 483.148,A -85,B 0,C 180,E1 -15638.912,E2 -15638.912} C_VEL
LIN {X 0,Y 312.627,Z 483.166,A -85,B 0,C 180,E1 -15641.656,E2 -15641.656} C_VEL
LIN {X 0,Y 312.683,Z 483.158,A -85,B 0,C 180,E1 -15645.686,E2 -15645.686} C_VEL
LIN {X 0,Y 312.693,Z 483.153,A -85,B 0,C 180,E1 -15649.642,E2 -15649.642} C_VEL
LIN {X 0,Y 312.861,Z 483.136,A -85,B 0,C 180,E1 -15652.254,E2 -15652.254} C_VEL
LIN {X 0,Y 312.71,Z 483.153,A -85,B 0,C 180,E1 -15654.842,E2 -15654.842} C_VEL
LIN {X 0,Y 312.982,Z 483.113,A -85,B 0,C 180,E1 -15658.714,E2 -15658.714} C_VEL
LIN {X 0,Y 313.11,Z 483.103,A -85,B 0,C 180,E1 -15660,E2 -15660} C_VEL
LIN {X 0,Y 312.928,Z 483.122,A -85,B 0,C 180,E1 -15662.575,E2 -15662.575} C_VEL
LIN {X 0,Y 312.883,Z 483.135,A -85,B 0,C 180,E1 -15666.651,E2 -15666.651} C_VEL
LIN {X 0,Y 312.777,Z 483.141,A -85,B 0,C 180,E1 -15669.05,E2 -15669.05} C_VEL
LIN {X 0,Y 312.626,Z 483.157,A -85,B 0,C 180,E1 -15672.992,E2 -15672.992} C_VEL
LIN {X 0,Y 312.628,Z 483.167,A -85,B 0,C 180,E1 -15675.65,E2 -15675.65} C_VEL
LIN {X 0,Y 312.621,Z 483.167,A -85,B 0,C 180,E1 -15679.238,E2 -15679.238} C_VEL
LIN {X 0,Y 312.536,Z 483.173,A -85,B 0,C 180,E1 -15682.79,E2 -15682.79} C_VEL
LIN {X 0,Y 312.593,Z 483.166,A -85,B 0,C 180,E1 -15685.937,E2 -15685.937} C_VEL
LIN {X 0,Y 312.541,Z 483.174,A -85,B 0,C 180,E1 -15689.651,E2 -15689.651} C_VEL
LIN {X 0,Y 312.513,Z 483.175,A -85,B 0,C 180,E1 -15693.691,E2 -15693.691} C_VEL
LIN {X 0,Y 312.533,Z 483.174,A -85,B 0,C 180,E1 -15697.384,E2 -15697.384} C_VEL
LIN {X 0,Y 312.495,Z 483.182,A -85,B 0,C 180,E1 -15700.709,E2 -15700.709} C_VEL
LIN {X 0,Y 312.524,Z 483.182,A -85,B 0,C 180,E1 -15704.197,E2 -15704.197} C_VEL
LIN {X 0,Y 312.543,Z 483.177,A -85,B 0,C 180,E1 -15707.907,E2 -15707.907} C_VEL
LIN {X 0,Y 312.553,Z 483.171,A -85,B 0,C 180,E1 -15711.907,E2 -15711.907} C_VEL
LIN {X 0,Y 312.56,Z 483.299,A -85,B 0,C 180,E1 -15712.99,E2 -15712.99} C_VEL
LIN {X 0,Y 315.784,Z 495.298,A -85,B 0,C 180,E1 -15716.96,E2 -15716.96} C_VEL
LIN {X 0,Y 318.576,Z 507.315,A -85,B 0,C 180,E1 -15720.629,E2 -15720.629} C_VEL
LIN {X 0,Y 320.115,Z 515.234,A -85,B 0,C 180,E1 -15722.901,E2 -15722.901} C_VEL
LIN {X 0,Y 320.156,Z 517.074,A -85,B 0,C 180,E1 -15723.39,E2 -15723.39} C_VEL
LIN {X 0,Y 325.879,Z 545.099,A -85,B 0,C 180,E1 -15724.579,E2 -15724.579} C_VEL
LIN {X 0,Y 327.258,Z 553.101,A -85,B 0,C 180,E1 -15724.882,E2 -15724.882} C_VEL
LIN {X 0,Y 325.491,Z 633.11,A -85,B 0,C 180,E1 -15726.542,E2 -15726.542} C_VEL
LIN {X 0,Y 324.884,Z 645.765,A -85,B 0,C 180,E1 -15727.044,E2 -15727.044} C_VEL
LIN {X 0,Y 323.863,Z 658.213,A -85,B 0,C 180,E1 -15727.767,E2 -15727.767} C_VEL
LIN {X 0,Y 322.535,Z 670.733,A -85,B 0,C 180,E1 -15728.763,E2 -15728.763} C_VEL
LIN {X 0,Y 320.92,Z 682.465,A -85,B 0,C 180,E1 -15729.992,E2 -15729.992} C_VEL
LIN {X 0,Y 319.425,Z 692.876,A -85,B 0,C 180,E1 -15731.383,E2 -15731.383} C_VEL
LIN {X 0,Y 317.779,Z 702.464,A -85,B 0,C 180,E1 -15732.962,E2 -15732.962} C_VEL
LIN {X 0,Y 316.078,Z 711.709,A -85,B 0,C 180,E1 -15734.857,E2 -15734.857} C_VEL
LIN {X 0,Y 314.701,Z 719.118,A -85,B 0,C 180,E1 -15736.769,E2 -15736.769} C_VEL
LIN {X 0,Y 313.707,Z 724.224,A -85,B 0,C 180,E1 -15738.37,E2 -15738.37} C_VEL
LIN {X 0,Y 312.693,Z 729.215,A -85,B 0,C 180,E1 -15740.297,E2 -15740.297} C_VEL
LIN {X 0,Y 311.984,Z 733.402,A -85,B 0,C 180,E1 -15742.387,E2 -15742.387} C_VEL
LIN {X 0,Y 311.749,Z 735.206,A -85,B 0,C 180,E1 -15743.53,E2 -15743.53} C_VEL
LIN {X 0,Y 311.23,Z 738.128,A -85,B 0,C 180,E1 -15746.117,E2 -15746.117} C_VEL
LIN {X 0,Y 311.049,Z 739.592,A -85,B 0,C 180,E1 -15748.707,E2 -15748.707} C_VEL
LIN {X 0,Y 311.049,Z 739.628,A -85,B 0,C 180,E1 -15751.296,E2 -15751.296} C_VEL
LIN {X 0,Y 311.215,Z 738.213,A -85,B 0,C 180,E1 -15753.886,E2 -15753.886} C_VEL
LIN {X 0,Y 311.717,Z 735.348,A -85,B 0,C 180,E1 -15756.474,E2 -15756.474} C_VEL
LIN {X 0,Y 312.237,Z 732.126,A -85,B 0,C 180,E1 -15758.415,E2 -15758.415} C_VEL
LIN {X 0,Y 312.977,Z 727.916,A -85,B 0,C 180,E1 -15760.351,E2 -15760.351} C_VEL
LIN {X 0,Y 314.265,Z 721.615,A -85,B 0,C 180,E1 -15762.596,E2 -15762.596} C_VEL
LIN {X 0,Y 315.627,Z 714.763,A -85,B 0,C 180,E1 -15764.509,E2 -15764.509} C_VEL
LIN {X 0,Y 316.816,Z 707.849,A -85,B 0,C 180,E1 -15766.1,E2 -15766.1} C_VEL
LIN {X 0,Y 318.355,Z 699.523,A -85,B 0,C 180,E1 -15767.672,E2 -15767.672} C_VEL
LIN {X 0,Y 319.963,Z 689.317,A -85,B 0,C 180,E1 -15769.238,E2 -15769.238} C_VEL
LIN {X 0,Y 321.401,Z 679.273,A -85,B 0,C 180,E1 -15770.481,E2 -15770.481} C_VEL
LIN {X 0,Y 322.855,Z 668.344,A -85,B 0,C 180,E1 -15771.553,E2 -15771.553} C_VEL
LIN {X 0,Y 324.127,Z 656.267,A -85,B 0,C 180,E1 -15772.469,E2 -15772.469} C_VEL
LIN {X 0,Y 325.051,Z 643.035,A -85,B 0,C 180,E1 -15773.2,E2 -15773.2} C_VEL
LIN {X 0,Y 325.717,Z 629.615,A -85,B 0,C 180,E1 -15773.655,E2 -15773.655} C_VEL
LIN {X 0,Y 327.287,Z 552.317,A -85,B 0,C 180,E1 -15775.245,E2 -15775.245} C_VEL
LIN {X 0,Y 321.889,Z 524.804,A -85,B 0,C 180,E1 -15776.371,E2 -15776.371} C_VEL
LIN {X 0,Y 320.148,Z 516.949,A -85,B 0,C 180,E1 -15776.76,E2 -15776.76} C_VEL
LIN {X 0,Y 319.563,Z 512.25,A -85,B 0,C 180,E1 -15778.061,E2 -15778.061} C_VEL
LIN {X 0,Y 317.111,Z 500.975,A -85,B 0,C 180,E1 -15781.389,E2 -15781.389} C_VEL
LIN {X 0,Y 314.832,Z 491.731,A -85,B 0,C 180,E1 -15784.314,E2 -15784.314} C_VEL
LIN {X 0,Y 314.555,Z 490.703,A -85,B 0,C 180,E1 -15784.652,E2 -15784.652} C_VEL
LIN {X 0,Y 313.335,Z 489.294,A -85,B 0,C 180,E1 -15785.268,E2 -15785.268} C_VEL
LIN {X 0,Y 306.545,Z 486.117,A -85,B 0,C 180,E1 -15787.16,E2 -15787.16} C_VEL
LIN {X 0,Y 305.594,Z 484.73,A -85,B 0,C 180,E1 -15787.737,E2 -15787.737} C_VEL
LIN {X 0,Y 305.497,Z 484.053,A -85,B 0,C 180,E1 -15787.997,E2 -15787.997} C_VEL
LIN {X 0,Y 305.447,Z 484.059,A -85,B 0,C 180,E1 -15791.858,E2 -15791.858} C_VEL
LIN {X 0,Y 305.407,Z 484.065,A -85,B 0,C 180,E1 -15795.512,E2 -15795.512} C_VEL
LIN {X 0,Y 305.447,Z 484.052,A -85,B 0,C 180,E1 -15798.144,E2 -15798.144} C_VEL
LIN {X 0,Y 305.474,Z 484.046,A -85,B 0,C 180,E1 -15801.597,E2 -15801.597} C_VEL
LIN {X 0,Y 305.469,Z 484.059,A -85,B 0,C 180,E1 -15804.887,E2 -15804.887} C_VEL
LIN {X 0,Y 305.517,Z 484.198,A -85,B 0,C 180,E1 -15806.735,E2 -15806.735} C_VEL
LIN {X 0,Y 309.455,Z 501.14,A -85,B 0,C 180,E1 -15810.398,E2 -15810.398} C_VEL
LIN {X 0,Y 311.487,Z 510.93,A -85,B 0,C 180,E1 -15812.46,E2 -15812.46} C_VEL
LIN {X 0,Y 311.241,Z 518.226,A -85,B 0,C 180,E1 -15813.875,E2 -15813.875} C_VEL
LIN {X 0,Y 310.152,Z 532.929,A -85,B 0,C 180,E1 -15816.668,E2 -15816.668} C_VEL
LIN {X 0,Y 313.212,Z 558.9,A -85,B 0,C 180,E1 -15817.711,E2 -15817.711} C_VEL
LIN {X 0,Y 310.276,Z 645.718,A -85,B 0,C 180,E1 -15820.568,E2 -15820.568} C_VEL
LIN {X 0,Y 309.6,Z 659.555,A -85,B 0,C 180,E1 -15821.298,E2 -15821.298} C_VEL
LIN {X 0,Y 308.902,Z 672.927,A -85,B 0,C 180,E1 -15822.284,E2 -15822.284} C_VEL
LIN {X 0,Y 307.992,Z 685.53,A -85,B 0,C 180,E1 -15823.51,E2 -15823.51} C_VEL
LIN {X 0,Y 307.078,Z 696.897,A -85,B 0,C 180,E1 -15824.91,E2 -15824.91} C_VEL
LIN {X 0,Y 306.274,Z 706.675,A -85,B 0,C 180,E1 -15826.396,E2 -15826.396} C_VEL
LIN {X 0,Y 305.498,Z 715.675,A -85,B 0,C 180,E1 -15828.051,E2 -15828.051} C_VEL
LIN {X 0,Y 304.931,Z 723.146,A -85,B 0,C 180,E1 -15829.71,E2 -15829.71} C_VEL
LIN {X 0,Y 304.393,Z 730.441,A -85,B 0,C 180,E1 -15831.703,E2 -15831.703} C_VEL
LIN {X 0,Y 304.101,Z 736.034,A -85,B 0,C 180,E1 -15833.606,E2 -15833.606} C_VEL
LIN {X 0,Y 303.885,Z 741.478,A -85,B 0,C 180,E1 -15836.021,E2 -15836.021} C_VEL
LIN {X 0,Y 303.764,Z 743.714,A -85,B 0,C 180,E1 -15837.348,E2 -15837.348} C_VEL
LIN {X 0,Y 303.712,Z 745.507,A -85,B 0,C 180,E1 -15838.674,E2 -15838.674} C_VEL
LIN {X 0,Y 303.722,Z 746.842,A -85,B 0,C 180,E1 -15840,E2 -15840} C_VEL
LIN {X 0,Y 303.844,Z 747.7,A -85,B 0,C 180,E1 -15841.325,E2 -15841.325} C_VEL
LIN {X 0,Y 304.015,Z 748.148,A -85,B 0,C 180,E1 -15842.65,E2 -15842.65} C_VEL
LIN {X 0,Y 304.159,Z 748.177,A -85,B 0,C 180,E1 -15843.975,E2 -15843.975} C_VEL
LIN {X 0,Y 304.34,Z 747.737,A -85,B 0,C 180,E1 -15845.3,E2 -15845.3} C_VEL
LIN {X 0,Y 304.718,Z 746.876,A -85,B 0,C 180,E1 -15846.622,E2 -15846.622} C_VEL
LIN {X 0,Y 305.387,Z 745.171,A -85,B 0,C 180,E1 -15848.272,E2 -15848.272} C_VEL
LIN {X 0,Y 306.454,Z 741.63,A -85,B 0,C 180,E1 -15850.572,E2 -15850.572} C_VEL
LIN {X 0,Y 307.68,Z 737.413,A -85,B 0,C 180,E1 -15852.533,E2 -15852.533} C_VEL
LIN {X 0,Y 309.153,Z 731.982,A -85,B 0,C 180,E1 -15854.481,E2 -15854.481} C_VEL
LIN {X 0,Y 311.347,Z 723.851,A -85,B 0,C 180,E1 -15856.726,E2 -15856.726} C_VEL
LIN {X 0,Y 313.154,Z 716.713,A -85,B 0,C 180,E1 -15858.312,E2 -15858.312} C_VEL
LIN {X 0,Y 315.11,Z 708.453,A -85,B 0,C 180,E1 -15859.824,E2 -15859.824} C_VEL
LIN {X 0,Y 317.261,Z 698.478,A -85,B 0,C 180,E1 -15861.31,E2 -15861.31} C_VEL
LIN {X 0,Y 319.356,Z 687.527,A -85,B 0,C 180,E1 -15862.651,E2 -15862.651} C_VEL
LIN {X 0,Y 321.171,Z 676.718,A -85,B 0,C 180,E1 -15863.709,E2 -15863.709} C_VEL
LIN {X 0,Y 323.16,Z 662.771,A -85,B 0,C 180,E1 -15864.749,E2 -15864.749} C_VEL
LIN {X 0,Y 324.651,Z 649.312,A -85,B 0,C 180,E1 -15865.483,E2 -15865.483} C_VEL
LIN {X 0,Y 332.694,Z 567.703,A -85,B 0,C 180,E1 -15868.631,E2 -15868.631} C_VEL
LIN {X 0,Y 331.151,Z 556.768,A -85,B 0,C 180,E1 -15869.651,E2 -15869.651} C_VEL
LIN {X 0,Y 328.639,Z 542.672,A -85,B 0,C 180,E1 -15871.238,E2 -15871.238} C_VEL
LIN {X 0,Y 327.998,Z 539.502,A -85,B 0,C 180,E1 -15871.723,E2 -15871.723} C_VEL
LIN {X 0,Y 327.345,Z 532.91,A -85,B 0,C 180,E1 -15873.932,E2 -15873.932} C_VEL
LIN {X 0,Y 326.512,Z 527.382,A -85,B 0,C 180,E1 -15876.17,E2 -15876.17} C_VEL
LIN {X 0,Y 325.411,Z 522.067,A -85,B 0,C 180,E1 -15878.966,E2 -15878.966} C_VEL
LIN {X 0,Y 324.855,Z 519.568,A -85,B 0,C 180,E1 -15880.78,E2 -15880.78} C_VEL
LIN {X 0,Y 324.448,Z 517.766,A -85,B 0,C 180,E1 -15882.565,E2 -15882.565} C_VEL
LIN {X 0,Y 324.303,Z 516.728,A -85,B 0,C 180,E1 -15884.343,E2 -15884.343} C_VEL
LIN {X 0,Y 324.424,Z 516.32,A -85,B 0,C 180,E1 -15886.113,E2 -15886.113} C_VEL
LIN {X 0,Y 324.949,Z 516.568,A -85,B 0,C 180,E1 -15887.895,E2 -15887.895} C_VEL
LIN {X 0,Y 325.848,Z 517.47,A -85,B 0,C 180,E1 -15889.679,E2 -15889.679} C_VEL
LIN {X 0,Y 327.177,Z 519.103,A -85,B 0,C 180,E1 -15891.467,E2 -15891.467} C_VEL
LIN {X 0,Y 328.047,Z 520.404,A -85,B 0,C 180,E1 -15892.437,E2 -15892.437} C_VEL
LIN {X 0,Y 328.384,Z 524.033,A -85,B 0,C 180,E1 -15893.657,E2 -15893.657} C_VEL
LIN {X 0,Y 329.603,Z 533.997,A -85,B 0,C 180,E1 -15896.262,E2 -15896.262} C_VEL
LIN {X 0,Y 330.257,Z 538.089,A -85,B 0,C 180,E1 -15897.168,E2 -15897.168} C_VEL
LIN {X 0,Y 330.322,Z 540.34,A -85,B 0,C 180,E1 -15897.539,E2 -15897.539} C_VEL
LIN {X 0,Y 329.641,Z 547.603,A -85,B 0,C 180,E1 -15898.437,E2 -15898.437} C_VEL
LIN {X 0,Y 329.266,Z 552.079,A -85,B 0,C 180,E1 -15898.86,E2 -15898.86} C_VEL
LIN {X 0,Y 329.359,Z 562.287,A -85,B 0,C 180,E1 -15899.583,E2 -15899.583} C_VEL
LIN {X 0,Y 320.062,Z 650.63,A -85,B 0,C 180,E1 -15903.113,E2 -15903.113} C_VEL
LIN {X 0,Y 318.196,Z 672.37,A -85,B 0,C 180,E1 -15904.048,E2 -15904.048} C_VEL
LIN {X 0,Y 316.819,Z 686.377,A -85,B 0,C 180,E1 -15904.895,E2 -15904.895} C_VEL
LIN {X 0,Y 315.385,Z 697.964,A -85,B 0,C 180,E1 -15905.827,E2 -15905.827} C_VEL
LIN {X 0,Y 313.805,Z 709.455,A -85,B 0,C 180,E1 -15906.982,E2 -15906.982} C_VEL
LIN {X 0,Y 312.165,Z 720.647,A -85,B 0,C 180,E1 -15908.365,E2 -15908.365} C_VEL
LIN {X 0,Y 310.432,Z 730.299,A -85,B 0,C 180,E1 -15909.801,E2 -15909.801} C_VEL
LIN {X 0,Y 308.565,Z 740.997,A -85,B 0,C 180,E1 -15911.748,E2 -15911.748} C_VEL
LIN {X 0,Y 307.085,Z 749.65,A -85,B 0,C 180,E1 -15913.717,E2 -15913.717} C_VEL
LIN {X 0,Y 305.934,Z 756.775,A -85,B 0,C 180,E1 -15915.701,E2 -15915.701} C_VEL
LIN {X 0,Y 304.803,Z 763.419,A -85,B 0,C 180,E1 -15918.021,E2 -15918.021} C_VEL
LIN {X 0,Y 304.212,Z 767.818,A -85,B 0,C 180,E1 -15920.021,E2 -15920.021} C_VEL
LIN {X 0,Y 303.864,Z 771.126,A -85,B 0,C 180,E1 -15922.022,E2 -15922.022} C_VEL
LIN {X 0,Y 303.695,Z 773.653,A -85,B 0,C 180,E1 -15924.32,E2 -15924.32} C_VEL
LIN {X 0,Y 303.731,Z 774.707,A -85,B 0,C 180,E1 -15926.018,E2 -15926.018} C_VEL
LIN {X 0,Y 303.9,Z 775.283,A -85,B 0,C 180,E1 -15929.998,E2 -15929.998} C_VEL
LIN {X 0,Y 303.828,Z 775.088,A -85,B 0,C 180,E1 -15931.324,E2 -15931.324} C_VEL
LIN {X 0,Y 303.763,Z 773.593,A -85,B 0,C 180,E1 -15933.978,E2 -15933.978} C_VEL
LIN {X 0,Y 303.816,Z 770.614,A -85,B 0,C 180,E1 -15936.64,E2 -15936.64} C_VEL
LIN {X 0,Y 303.998,Z 766.072,A -85,B 0,C 180,E1 -15939.311,E2 -15939.311} C_VEL
LIN {X 0,Y 304.423,Z 761.54,A -85,B 0,C 180,E1 -15941.315,E2 -15941.315} C_VEL
LIN {X 0,Y 305.264,Z 754.929,A -85,B 0,C 180,E1 -15943.648,E2 -15943.648} C_VEL
LIN {X 0,Y 306.054,Z 749.171,A -85,B 0,C 180,E1 -15945.322,E2 -15945.322} C_VEL
LIN {X 0,Y 307.344,Z 741.056,A -85,B 0,C 180,E1 -15947.292,E2 -15947.292} C_VEL
LIN {X 0,Y 308.935,Z 731.175,A -85,B 0,C 180,E1 -15949.258,E2 -15949.258} C_VEL
LIN {X 0,Y 310.845,Z 720.186,A -85,B 0,C 180,E1 -15951.032,E2 -15951.032} C_VEL
LIN {X 0,Y 312.691,Z 708.002,A -85,B 0,C 180,E1 -15952.63,E2 -15952.63} C_VEL
LIN {X 0,Y 314.434,Z 695.813,A -85,B 0,C 180,E1 -15953.896,E2 -15953.896} C_VEL
LIN {X 0,Y 316.079,Z 682.284,A -85,B 0,C 180,E1 -15954.988,E2 -15954.988} C_VEL
LIN {X 0,Y 317.487,Z 668.116,A -85,B 0,C 180,E1 -15955.835,E2 -15955.835} C_VEL
LIN {X 0,Y 318.534,Z 654.161,A -85,B 0,C 180,E1 -15956.403,E2 -15956.403} C_VEL
LIN {X 0,Y 320.369,Z 596.106,A -85,B 0,C 180,E1 -15957.805,E2 -15957.805} C_VEL
LIN {X 0,Y 321.373,Z 558.631,A -85,B 0,C 180,E1 -15958.694,E2 -15958.694} C_VEL
LIN {X 0,Y 316.821,Z 526.516,A -85,B 0,C 180,E1 -15959.958,E2 -15959.958} C_VEL
LIN {X 0,Y 315.96,Z 523.443,A -85,B 0,C 180,E1 -15960.124,E2 -15960.124} C_VEL
LIN {X 0,Y 315.22,Z 521.346,A -85,B 0,C 180,E1 -15960.299,E2 -15960.299} C_VEL
LIN {X 0,Y 312.65,Z 509.822,A -85,B 0,C 180,E1 -15963.288,E2 -15963.288} C_VEL
LIN {X 0,Y 309.616,Z 498.129,A -85,B 0,C 180,E1 -15966.515,E2 -15966.515} C_VEL
LIN {X 0,Y 306.579,Z 487.655,A -85,B 0,C 180,E1 -15969.627,E2 -15969.627} C_VEL
LIN {X 0,Y 305.487,Z 484.057,A -85,B 0,C 180,E1 -15970.791,E2 -15970.791} C_VEL
LIN {X 0,Y 305.537,Z 484.051,A -85,B 0,C 180,E1 -15974.515,E2 -15974.515} C_VEL
LIN {X 0,Y 305.494,Z 484.05,A -85,B 0,C 180,E1 -15978.152,E2 -15978.152} C_VEL
LIN {X 0,Y 305.512,Z 484.049,A -85,B 0,C 180,E1 -15981.603,E2 -15981.603} C_VEL
LIN {X 0,Y 305.454,Z 484.035,A -85,B 0,C 180,E1 -15984.886,E2 -15984.886} C_VEL
LIN {X 0,Y 305.446,Z 484.055,A -85,B 0,C 180,E1 -15988.353,E2 -15988.353} C_VEL
LIN {X 0,Y 305.511,Z 484.051,A -85,B 0,C 180,E1 -15991.113,E2 -15991.113} C_VEL
LIN {X 0,Y 305.562,Z 484.048,A -85,B 0,C 180,E1 -15994.087,E2 -15994.087} C_VEL
LIN {X 0,Y 305.472,Z 484.022,A -85,B 0,C 180,E1 -15998.401,E2 -15998.401} C_VEL
LIN {X 0,Y 305.569,Z 484.047,A -85,B 0,C 180,E1 -16001.216,E2 -16001.216} C_VEL
LIN {X 0,Y 305.638,Z 484.036,A -85,B 0,C 180,E1 -16005.349,E2 -16005.349} C_VEL
LIN {X 0,Y 305.63,Z 484.032,A -85,B 0,C 180,E1 -16009.4,E2 -16009.4} C_VEL
LIN {X 0,Y 305.802,Z 484.017,A -85,B 0,C 180,E1 -16012.074,E2 -16012.074} C_VEL
LIN {X 0,Y 305.681,Z 484.027,A -85,B 0,C 180,E1 -16014.724,E2 -16014.724} C_VEL
LIN {X 0,Y 305.948,Z 483.989,A -85,B 0,C 180,E1 -16018.684,E2 -16018.684} C_VEL
LIN {X 0,Y 305.948,Z 483.998,A -85,B 0,C 180,E1 -16021.316,E2 -16021.316} C_VEL
LIN {X 0,Y 305.842,Z 484.012,A -85,B 0,C 180,E1 -16026.598,E2 -16026.598} C_VEL
LIN {X 0,Y 305.725,Z 484.021,A -85,B 0,C 180,E1 -16029.26,E2 -16029.26} C_VEL
LIN {X 0,Y 305.58,Z 484.034,A -85,B 0,C 180,E1 -16033.297,E2 -16033.297} C_VEL
LIN {X 0,Y 305.584,Z 484.046,A -85,B 0,C 180,E1 -16036.021,E2 -16036.021} C_VEL
LIN {X 0,Y 305.567,Z 484.046,A -85,B 0,C 180,E1 -16039.446,E2 -16039.446} C_VEL
LIN {X 0,Y 305.481,Z 484.053,A -85,B 0,C 180,E1 -16043.042,E2 -16043.042} C_VEL
LIN {X 0,Y 305.539,Z 484.043,A -85,B 0,C 180,E1 -16046.229,E2 -16046.229} C_VEL
LIN {X 0,Y 305.495,Z 484.053,A -85,B 0,C 180,E1 -16049.054,E2 -16049.054} C_VEL
LIN {X 0,Y 305.441,Z 484.062,A -85,B 0,C 180,E1 -16051.953,E2 -16051.953} C_VEL
LIN {X 0,Y 305.457,Z 484.062,A -85,B 0,C 180,E1 -16055.114,E2 -16055.114} C_VEL
LIN {X 0,Y 305.475,Z 484.06,A -85,B 0,C 180,E1 -16058.538,E2 -16058.538} C_VEL
LIN {X 0,Y 305.491,Z 484.055,A -85,B 0,C 180,E1 -16062.596,E2 -16062.596} C_VEL
LIN {X 0,Y 305.486,Z 484.057,A -85,B 0,C 180,E1 -16066.359,E2 -16066.359} C_VEL
LIN {X 0,Y 305.494,Z 484.055,A -85,B 0,C 180,E1 -16069.901,E2 -16069.901} C_VEL
LIN {X 0,Y 305.525,Z 484.092,A -85,B 0,C 180,E1 -16072.183,E2 -16072.183} C_VEL
LIN {X 0,Y 308.581,Z 495.494,A -85,B 0,C 180,E1 -16076.085,E2 -16076.085} C_VEL
LIN {X 0,Y 311.179,Z 506.267,A -85,B 0,C 180,E1 -16079.507,E2 -16079.507} C_VEL
LIN {X 0,Y 313.35,Z 517.069,A -85,B 0,C 180,E1 -16082.701,E2 -16082.701} C_VEL
LIN {X 0,Y 315.108,Z 523.835,A -85,B 0,C 180,E1 -16083.062,E2 -16083.062} C_VEL
LIN {X 0,Y 320.477,Z 551.088,A -85,B 0,C 180,E1 -16084.224,E2 -16084.224} C_VEL
LIN {X 0,Y 320.958,Z 554.589,A -85,B 0,C 180,E1 -16084.349,E2 -16084.349} C_VEL
LIN {X 0,Y 319.095,Z 633.001,A -85,B 0,C 180,E1 -16086,E2 -16086} C_VEL
LIN {X 0,Y 318.448,Z 645.782,A -85,B 0,C 180,E1 -16086.509,E2 -16086.509} C_VEL
LIN {X 0,Y 317.321,Z 658.867,A -85,B 0,C 180,E1 -16087.284,E2 -16087.284} C_VEL
LIN {X 0,Y 315.97,Z 671.293,A -85,B 0,C 180,E1 -16088.3,E2 -16088.3} C_VEL
LIN {X 0,Y 314.29,Z 682.967,A -85,B 0,C 180,E1 -16089.551,E2 -16089.551} C_VEL
LIN {X 0,Y 312.677,Z 693.662,A -85,B 0,C 180,E1 -16091.017,E2 -16091.017} C_VEL
LIN {X 0,Y 311.033,Z 702.917,A -85,B 0,C 180,E1 -16092.581,E2 -16092.581} C_VEL
LIN {X 0,Y 309.246,Z 712.145,A -85,B 0,C 180,E1 -16094.514,E2 -16094.514} C_VEL
LIN {X 0,Y 307.821,Z 719.543,A -85,B 0,C 180,E1 -16096.468,E2 -16096.468} C_VEL
LIN {X 0,Y 306.789,Z 724.646,A -85,B 0,C 180,E1 -16098.104,E2 -16098.104} C_VEL
LIN {X 0,Y 305.711,Z 729.633,A -85,B 0,C 180,E1 -16100.073,E2 -16100.073} C_VEL
LIN {X 0,Y 304.921,Z 734.044,A -85,B 0,C 180,E1 -16102.348,E2 -16102.348} C_VEL
LIN {X 0,Y 304.359,Z 737.269,A -85,B 0,C 180,E1 -16104.702,E2 -16104.702} C_VEL
LIN {X 0,Y 304.063,Z 739.444,A -85,B 0,C 180,E1 -16107.352,E2 -16107.352} C_VEL
LIN {X 0,Y 303.948,Z 740.207,A -85,B 0,C 180,E1 -16110.002,E2 -16110.002} C_VEL
LIN {X 0,Y 304.058,Z 739.504,A -85,B 0,C 180,E1 -16112.651,E2 -16112.651} C_VEL
LIN {X 0,Y 304.341,Z 737.377,A -85,B 0,C 180,E1 -16115.302,E2 -16115.302} C_VEL
LIN {X 0,Y 304.956,Z 734.135,A -85,B 0,C 180,E1 -16117.701,E2 -16117.701} C_VEL
LIN {X 0,Y 305.708,Z 729.875,A -85,B 0,C 180,E1 -16119.93,E2 -16119.93} C_VEL
LIN {X 0,Y 306.733,Z 724.944,A -85,B 0,C 180,E1 -16121.902,E2 -16121.902} C_VEL
LIN {X 0,Y 307.958,Z 718.802,A -85,B 0,C 180,E1 -16123.866,E2 -16123.866} C_VEL
LIN {X 0,Y 309.186,Z 712.568,A -85,B 0,C 180,E1 -16125.492,E2 -16125.492} C_VEL
LIN {X 0,Y 310.682,Z 705.122,A -85,B 0,C 180,E1 -16127.104,E2 -16127.104} C_VEL
LIN {X 0,Y 312.392,Z 695.756,A -85,B 0,C 180,E1 -16128.771,E2 -16128.771} C_VEL
LIN {X 0,Y 313.968,Z 685.054,A -85,B 0,C 180,E1 -16130.303,E2 -16130.303} C_VEL
LIN {X 0,Y 315.672,Z 673.87,A -85,B 0,C 180,E1 -16131.554,E2 -16131.554} C_VEL
LIN {X 0,Y 317.206,Z 661.331,A -85,B 0,C 180,E1 -16132.643,E2 -16132.643} C_VEL
LIN {X 0,Y 318.28,Z 648.526,A -85,B 0,C 180,E1 -16133.464,E2 -16133.464} C_VEL
LIN {X 0,Y 319.058,Z 635.983,A -85,B 0,C 180,E1 -16134.007,E2 -16134.007} C_VEL
